C09149=1177.909,-61.811,-42.425,179.391,5.754,149.202
C09150=1177.904,-61.560,-42.436,179.394,5.755,149.202
C09151=1177.898,-61.311,-42.447,179.396,5.754,149.201
C09152=1177.894,-61.062,-42.458,179.398,5.755,149.201
C09153=1177.888,-60.811,-42.470,179.400,5.756,149.200
C09154=1177.883,-60.562,-42.481,179.403,5.756,149.199
C09155=1177.878,-60.313,-42.492,179.405,5.756,149.199
C09156=1177.872,-60.062,-42.503,179.407,5.756,149.198
C09157=1177.867,-59.813,-42.514,179.410,5.757,149.198
C09158=1177.862,-59.564,-42.525,179.412,5.757,149.197
C09159=1177.857,-59.314,-42.537,179.414,5.757,149.196
C09160=1177.851,-59.064,-42.547,179.417,5.758,149.196
C09161=1177.847,-58.815,-42.559,179.419,5.758,149.195
C09162=1177.841,-58.565,-42.570,179.421,5.758,149.194
C09163=1177.836,-58.314,-42.581,179.423,5.759,149.194
C09164=1177.831,-58.065,-42.592,179.426,5.759,149.193
C09165=1177.825,-57.815,-42.604,179.429,5.760,149.193
C09166=1177.821,-57.566,-42.615,179.430,5.760,149.192
C09167=1177.815,-57.316,-42.625,179.433,5.760,149.191
C09168=1177.810,-57.066,-42.637,179.436,5.761,149.191
C09169=1177.805,-56.817,-42.649,179.437,5.761,149.190
C09170=1177.800,-56.567,-42.660,179.440,5.761,149.189
C09171=1177.794,-56.318,-42.671,179.442,5.762,149.189
C09172=1177.789,-56.068,-42.682,179.445,5.762,149.188
C09173=1177.784,-55.818,-42.694,179.447,5.762,149.188
C09174=1177.779,-55.568,-42.705,179.449,5.763,149.187
C09175=1177.773,-55.319,-42.717,179.452,5.763,149.186
C09176=1177.768,-55.069,-42.728,179.454,5.763,149.186
C09177=1177.763,-54.819,-42.738,179.456,5.763,149.185
C09178=1177.758,-54.569,-42.750,179.459,5.764,149.185
C09179=1177.753,-54.320,-42.761,179.461,5.764,149.184
C09180=1177.747,-54.070,-42.773,179.464,5.765,149.183
C09181=1177.743,-53.821,-42.784,179.466,5.765,149.183
C09182=1177.737,-53.571,-42.796,179.468,5.765,149.182
C09183=1177.732,-53.322,-42.807,179.470,5.766,149.181
C09184=1177.726,-53.072,-42.819,179.473,5.766,149.181
C09185=1177.721,-52.821,-42.830,179.475,5.766,149.180
C09186=1177.717,-52.572,-42.841,179.477,5.767,149.180
C09187=1177.711,-52.322,-42.853,179.480,5.767,149.179
C09188=1177.706,-52.073,-42.864,179.482,5.767,149.178
C09189=1177.701,-51.823,-42.876,179.484,5.768,149.178
C09190=1177.696,-51.573,-42.887,179.487,5.768,149.177
C09191=1177.690,-51.324,-42.899,179.489,5.769,149.177
C09192=1177.686,-51.074,-42.910,179.492,5.769,149.176
C09193=1177.680,-50.825,-42.922,179.494,5.769,149.175
C09194=1177.674,-50.575,-42.934,179.496,5.770,149.175
C09195=1177.670,-50.325,-42.945,179.499,5.770,149.174
C09196=1177.664,-50.054,-42.957,179.501,5.771,149.173
C09197=1177.658,-49.784,-42.970,179.504,5.771,149.173
C09198=1177.652,-49.513,-42.982,179.506,5.771,149.172
C09199=1177.647,-49.244,-42.995,179.508,5.772,149.171
C09200=1177.642,-48.994,-43.006,179.511,5.772,149.171
C09201=1177.636,-48.744,-43.018,179.514,5.772,149.170
C09202=1177.631,-48.494,-43.030,179.516,5.773,149.169
C09203=1177.626,-48.245,-43.041,179.518,5.773,149.169
C09204=1177.621,-47.995,-43.053,179.521,5.773,149.168
C09205=1177.616,-47.746,-43.064,179.523,5.774,149.168
C09206=1177.610,-47.496,-43.076,179.525,5.774,149.167
C09207=1177.605,-47.246,-43.088,179.528,5.775,149.166
C09208=1177.600,-46.996,-43.099,179.530,5.775,149.166
C09209=1177.595,-46.746,-43.111,179.532,5.775,149.165
C09210=1177.590,-46.497,-43.122,179.535,5.776,149.164
C09211=1177.585,-46.247,-43.135,179.537,5.777,149.164
C09212=1177.579,-45.998,-43.146,179.539,5.776,149.163
C09213=1177.574,-45.749,-43.157,179.542,5.777,149.162
C09214=1177.569,-45.499,-43.169,179.544,5.777,149.162
C09215=1177.563,-45.249,-43.181,179.547,5.778,149.161
C09216=1177.559,-44.999,-43.192,179.549,5.778,149.161
C09217=1177.553,-44.749,-43.204,179.551,5.778,149.160
C09218=1177.548,-44.500,-43.216,179.554,5.779,149.159
C09219=1177.543,-44.250,-43.228,179.556,5.780,149.159
C09220=1177.538,-44.000,-43.240,179.559,5.780,149.158
C09221=1177.533,-43.751,-43.251,179.561,5.780,149.158
C09222=1177.527,-43.501,-43.263,179.563,5.780,149.157
C09223=1177.522,-43.251,-43.275,179.565,5.781,149.156
C09224=1177.516,-43.002,-43.287,179.568,5.781,149.156
C09225=1177.512,-42.753,-43.299,179.570,5.782,149.155
C09226=1177.506,-42.503,-43.311,179.572,5.782,149.154
C09227=1177.501,-42.253,-43.322,179.575,5.782,149.154
C09228=1177.496,-42.003,-43.334,179.577,5.783,149.153
C09229=1177.491,-41.753,-43.346,179.580,5.783,149.153
C09230=1177.486,-41.504,-43.358,179.583,5.784,149.152
C09231=1177.481,-41.254,-43.370,179.584,5.784,149.151
C09232=1177.476,-41.004,-43.381,179.587,5.784,149.151
C09233=1177.470,-40.754,-43.393,179.590,5.785,149.150
C09234=1177.465,-40.505,-43.406,179.592,5.786,149.150
C09235=1177.460,-40.255,-43.417,179.594,5.786,149.149
C09236=1177.455,-40.005,-43.429,179.596,5.786,149.148
C09237=1177.450,-39.755,-43.441,179.599,5.786,149.148
C09238=1177.444,-39.506,-43.454,179.601,5.787,149.147
C09239=1177.439,-39.257,-43.464,179.604,5.787,149.146
C09240=1177.434,-39.007,-43.476,179.606,5.788,149.146
C09241=1177.429,-38.758,-43.489,179.608,5.788,149.145
C09242=1177.423,-38.508,-43.501,179.611,5.788,149.144
C09243=1177.418,-38.258,-43.513,179.613,5.789,149.144
C09244=1177.413,-38.009,-43.525,179.616,5.789,149.143
C09245=1177.408,-37.759,-43.537,179.618,5.790,149.142
C09246=1177.402,-37.509,-43.549,179.620,5.790,149.142
C09247=1177.397,-37.260,-43.561,179.623,5.790,149.141
C09248=1177.392,-37.010,-43.573,179.625,5.791,149.141
C09249=1177.386,-36.760,-43.585,179.627,5.792,149.140
C09250=1177.382,-36.511,-43.597,179.630,5.792,149.139
C09251=1177.377,-36.261,-43.609,179.633,5.792,149.139
C09252=1177.372,-36.012,-43.621,179.634,5.792,149.138
C09253=1177.366,-35.762,-43.633,179.637,5.793,149.138
C09254=1177.361,-35.512,-43.645,179.640,5.793,149.137
C09255=1177.356,-35.263,-43.658,179.642,5.794,149.136
C09256=1177.351,-35.012,-43.669,179.645,5.795,149.136
C09257=1177.346,-34.763,-43.682,179.647,5.795,149.135
C09258=1177.341,-34.513,-43.694,179.649,5.795,149.135
C09259=1177.336,-34.264,-43.707,179.651,5.796,149.134
C09260=1177.330,-34.014,-43.718,179.654,5.796,149.133
C09261=1177.325,-33.764,-43.731,179.656,5.797,149.133
C09262=1177.320,-33.514,-43.743,179.659,5.797,149.132
C09263=1177.314,-33.265,-43.755,179.662,5.798,149.131
C09264=1177.309,-33.015,-43.767,179.663,5.798,149.131
C09265=1177.305,-32.766,-43.779,179.666,5.798,149.130
C09266=1177.299,-32.516,-43.791,179.669,5.799,149.129
C09267=1177.294,-32.266,-43.803,179.671,5.799,149.129
C09268=1177.289,-32.017,-43.816,179.673,5.800,149.128
C09269=1177.284,-31.768,-43.828,179.676,5.800,149.128
C09270=1177.278,-31.518,-43.840,179.678,5.800,149.127
C09271=1177.273,-31.268,-43.853,179.680,5.801,149.126
C09272=1177.268,-31.018,-43.865,179.683,5.801,149.126
C09273=1177.263,-30.769,-43.878,179.685,5.802,149.125
C09274=1177.258,-30.519,-43.890,179.688,5.802,149.125
C09275=1177.253,-30.269,-43.902,179.690,5.803,149.124
C09276=1177.247,-30.019,-43.914,179.693,5.804,149.123
C09277=1177.242,-29.770,-43.927,179.695,5.803,149.123
C09278=1177.237,-29.521,-43.939,179.697,5.804,149.122
C09279=1177.232,-29.271,-43.951,179.700,5.805,149.121
C09280=1177.226,-29.021,-43.964,179.702,5.805,149.121
C09281=1177.222,-28.771,-43.977,179.705,5.805,149.120
C09282=1177.217,-28.521,-43.989,179.707,5.806,149.120
C09283=1177.211,-28.272,-44.001,179.710,5.807,149.119
C09284=1177.206,-28.022,-44.013,179.712,5.806,149.118
C09285=1177.201,-27.773,-44.026,179.714,5.807,149.118
C09286=1177.196,-27.524,-44.038,179.717,5.808,149.117
C09287=1177.190,-27.274,-44.050,179.719,5.808,149.116
C09288=1177.186,-27.024,-44.063,179.721,5.809,149.116
C09289=1177.181,-26.774,-44.076,179.724,5.809,149.115
C09290=1177.175,-26.524,-44.088,179.727,5.810,149.114
C09291=1177.170,-26.275,-44.100,179.728,5.810,149.114
C09292=1177.165,-26.026,-44.113,179.731,5.810,149.113
C09293=1177.160,-25.776,-44.125,179.734,5.811,149.113
C09294=1177.155,-25.526,-44.138,179.736,5.812,149.112
C09295=1177.150,-25.276,-44.150,179.739,5.812,149.111
C09296=1177.145,-25.027,-44.163,179.741,5.812,149.111
C09297=1177.140,-24.778,-44.175,179.743,5.813,149.110
C09298=1177.133,-24.528,-44.188,179.746,5.814,149.110
C09299=1177.129,-24.278,-44.201,179.748,5.813,149.109
C09300=1177.123,-24.009,-44.214,179.751,5.814,149.108
C09301=1177.118,-23.739,-44.228,179.753,5.815,149.108
C09302=1177.112,-23.469,-44.241,179.756,5.816,149.107
C09303=1177.107,-23.199,-44.255,179.759,5.816,149.106
C09304=1177.102,-22.950,-44.267,179.761,5.816,149.106
C09305=1177.097,-22.700,-44.280,179.764,5.816,149.105
C09306=1177.091,-22.450,-44.293,179.766,5.817,149.104
C09307=1177.086,-22.200,-44.305,179.768,5.818,149.104
C09308=1177.081,-21.951,-44.318,179.771,5.818,149.103
C09309=1177.076,-21.702,-44.331,179.773,5.819,149.103
C09310=1177.071,-21.452,-44.344,179.776,5.819,149.102
C09311=1177.066,-21.202,-44.356,179.779,5.820,149.101
C09312=1177.060,-20.953,-44.369,179.781,5.821,149.101
C09313=1177.055,-20.703,-44.381,179.783,5.820,149.100
C09314=1177.050,-20.453,-44.394,179.785,5.821,149.099
C09315=1177.045,-20.203,-44.407,179.788,5.822,149.099
C09316=1177.040,-19.954,-44.419,179.790,5.822,149.098
C09317=1177.034,-19.704,-44.433,179.793,5.822,149.098
C09318=1177.029,-19.454,-44.446,179.795,5.823,149.097
C09319=1177.024,-19.205,-44.458,179.798,5.824,149.096
C09320=1177.019,-18.956,-44.471,179.800,5.824,149.096
C09321=1177.014,-18.706,-44.483,179.803,5.825,149.095
C09322=1177.009,-18.456,-44.497,179.805,5.825,149.094
C09323=1177.004,-18.207,-44.510,179.807,5.825,149.094
C09324=1176.999,-17.957,-44.522,179.810,5.826,149.093
C09325=1176.994,-17.707,-44.535,179.812,5.826,149.093
C09326=1176.988,-17.458,-44.548,179.815,5.827,149.092
C09327=1176.983,-17.208,-44.560,179.817,5.828,149.091
C09328=1176.978,-16.958,-44.573,179.820,5.828,149.091
C09329=1176.973,-16.709,-44.586,179.822,5.829,149.090
C09330=1176.967,-16.459,-44.599,179.825,5.829,149.090
C09331=1176.962,-16.210,-44.612,179.827,5.830,149.089
C09332=1176.958,-15.960,-44.625,179.830,5.830,149.088
C09333=1176.952,-15.711,-44.638,179.832,5.831,149.088
C09334=1176.947,-15.461,-44.651,179.835,5.832,149.087
C09335=1176.942,-15.211,-44.664,179.837,5.831,149.086
C09336=1176.937,-14.962,-44.677,179.839,5.832,149.086
C09337=1176.931,-14.712,-44.690,179.842,5.833,149.085
C09338=1176.927,-14.462,-44.703,179.844,5.833,149.085
C09339=1176.922,-14.213,-44.715,179.846,5.834,149.084
C09340=1176.916,-13.963,-44.729,179.849,5.834,149.083
C09341=1176.911,-13.713,-44.742,179.852,5.835,149.083
C09342=1176.906,-13.464,-44.754,179.854,5.836,149.082
C09343=1176.900,-13.214,-44.767,179.857,5.836,149.082
C09344=1176.896,-12.964,-44.780,179.859,5.836,149.081
C09345=1176.890,-12.715,-44.794,179.861,5.837,149.080
C09346=1176.886,-12.465,-44.807,179.864,5.838,149.080
C09347=1176.881,-12.216,-44.820,179.867,5.838,149.079
C09348=1176.875,-11.966,-44.833,179.869,5.839,149.079
C09349=1176.870,-11.716,-44.846,179.872,5.840,149.078
C09350=1176.865,-11.467,-44.859,179.874,5.840,149.077
C09351=1176.860,-11.217,-44.873,179.876,5.840,149.077
C09352=1176.855,-10.968,-44.885,179.878,5.840,149.076
C09353=1176.849,-10.718,-44.899,179.881,5.841,149.075
C09354=1176.845,-10.468,-44.912,179.883,5.842,149.075
C09355=1176.840,-10.219,-44.924,179.886,5.842,149.074
C09356=1176.835,-9.969,-44.938,179.889,5.843,149.073
C09357=1176.829,-9.720,-44.951,179.891,5.843,149.073
C09358=1176.824,-9.470,-44.964,179.893,5.844,149.072
C09359=1176.819,-9.220,-44.977,179.896,5.844,149.072
C09360=1176.814,-8.971,-44.991,179.898,5.845,149.071
C09361=1176.809,-8.721,-45.004,179.901,5.846,149.070
C09362=1176.804,-8.472,-45.017,179.904,5.846,149.070
C09363=1176.799,-8.222,-45.030,179.906,5.847,149.069
C09364=1176.794,-7.973,-45.044,179.908,5.847,149.069
C09365=1176.788,-7.723,-45.057,179.911,5.848,149.068
C09366=1176.783,-7.473,-45.070,179.913,5.849,149.067
C09367=1176.778,-7.224,-45.084,179.916,5.849,149.067
C09368=1176.773,-6.974,-45.097,179.919,5.850,149.066
C09369=1176.767,-6.725,-45.110,179.921,5.851,149.066
C09370=1176.763,-6.475,-45.124,179.923,5.851,149.065
C09371=1176.757,-6.226,-45.137,179.926,5.851,149.064
C09372=1176.753,-5.976,-45.150,179.929,5.852,149.063
C09373=1176.747,-5.727,-45.164,179.931,5.853,149.063
C09374=1176.743,-5.477,-45.177,179.934,5.853,149.062
C09375=1176.737,-5.227,-45.190,179.936,5.854,149.062
C09376=1176.733,-4.978,-45.203,179.938,5.854,149.061
C09377=1176.727,-4.728,-45.217,179.940,5.854,149.060
C09378=1176.722,-4.478,-45.230,179.943,5.855,149.060
C09379=1176.717,-4.229,-45.244,179.945,5.855,149.059
C09380=1176.712,-3.979,-45.257,179.948,5.856,149.059
C09381=1176.707,-3.730,-45.270,179.951,5.856,149.058
C09382=1176.701,-3.480,-45.284,179.953,5.857,149.057
C09383=1176.697,-3.231,-45.297,179.955,5.858,149.057
C09384=1176.691,-2.981,-45.311,179.958,5.858,149.056
C09385=1176.686,-2.731,-45.323,179.960,5.859,149.056
C09386=1176.681,-2.482,-45.338,179.963,5.859,149.055
C09387=1176.675,-2.232,-45.351,179.965,5.860,149.055
C09388=1176.671,-1.982,-45.365,179.968,5.861,149.054
C09389=1176.665,-1.733,-45.378,179.970,5.861,149.053
C09390=1176.660,-1.483,-45.392,179.972,5.862,149.053
C09391=1176.655,-1.234,-45.405,179.975,5.863,149.052
C09392=1176.650,-0.984,-45.419,179.978,5.863,149.051
C09393=1176.645,-0.735,-45.432,179.980,5.864,149.051
C09394=1176.640,-0.485,-45.446,179.983,5.864,149.050
C09395=1176.635,-0.235,-45.459,179.985,5.865,149.049
C09396=1176.630,0.014,-45.473,179.987,5.866,149.049
C09397=1176.625,0.264,-45.487,179.990,5.866,149.048
C09398=1176.619,0.513,-45.500,179.993,5.867,149.048
C09399=1176.615,0.763,-45.514,179.995,5.867,149.047
C09400=1176.609,1.012,-45.527,179.998,5.868,149.046
C09401=1176.604,1.262,-45.541,-180.000,5.868,149.046
C09402=1176.600,1.512,-45.554,-179.998,5.869,149.045
C09403=1176.594,1.761,-45.568,-179.995,5.870,149.045
C09404=1176.589,2.030,-45.583,-179.992,5.871,149.044
C09405=1176.583,2.300,-45.598,-179.989,5.871,149.043
C09406=1176.577,2.569,-45.613,-179.986,5.872,149.043
C09407=1176.572,2.838,-45.628,-179.984,5.872,149.042
C09408=1176.567,3.088,-45.641,-179.982,5.873,149.041
C09409=1176.562,3.337,-45.655,-179.979,5.874,149.041
C09410=1176.557,3.587,-45.669,-179.976,5.874,149.040
C09411=1176.552,3.837,-45.683,-179.974,5.875,149.040
C09412=1176.547,4.086,-45.696,-179.971,5.875,149.039
C09413=1176.542,4.335,-45.710,-179.969,5.876,149.038
C09414=1176.537,4.586,-45.724,-179.967,5.877,149.038
C09415=1176.531,4.835,-45.738,-179.964,5.877,149.037
C09416=1176.527,5.084,-45.751,-179.961,5.878,149.036
C09417=1176.521,5.333,-45.765,-179.959,5.878,149.036
C09418=1176.516,5.584,-45.779,-179.956,5.879,149.035
C09419=1176.511,5.833,-45.793,-179.954,5.879,149.035
C09420=1176.506,6.082,-45.806,-179.952,5.880,149.034
C09421=1176.501,6.332,-45.821,-179.949,5.881,149.033
C09422=1176.496,6.582,-45.834,-179.947,5.882,149.033
C09423=1176.490,6.831,-45.848,-179.944,5.883,149.032
C09424=1176.485,7.081,-45.862,-179.941,5.883,149.032
C09425=1176.481,7.330,-45.877,-179.939,5.884,149.031
C09426=1176.475,7.580,-45.889,-179.936,5.885,149.030
C09427=1176.470,7.829,-45.904,-179.933,5.885,149.030
C09428=1176.465,8.079,-45.918,-179.931,5.886,149.029
C09429=1176.461,8.329,-45.932,-179.929,5.886,149.029
C09430=1176.455,8.578,-45.946,-179.926,5.887,149.028
C09431=1176.450,8.828,-45.960,-179.924,5.888,149.027
C09432=1176.446,9.078,-45.973,-179.921,5.888,149.027
C09433=1176.440,9.327,-45.987,-179.919,5.889,149.026
C09434=1176.435,9.576,-46.001,-179.916,5.890,149.026
C09435=1176.430,9.826,-46.016,-179.914,5.890,149.025
C09436=1176.425,10.076,-46.030,-179.911,5.890,149.024
C09437=1176.420,10.325,-46.044,-179.909,5.891,149.024
C09438=1176.415,10.574,-46.058,-179.906,5.892,149.023
C09439=1176.410,10.824,-46.072,-179.904,5.892,149.022
C09440=1176.404,11.073,-46.086,-179.901,5.893,149.022
C09441=1176.399,11.324,-46.100,-179.899,5.894,149.021
C09442=1176.395,11.573,-46.114,-179.896,5.895,149.021
C09443=1176.390,11.823,-46.128,-179.893,5.896,149.020
C09444=1176.384,12.072,-46.142,-179.891,5.896,149.019
C09445=1176.379,12.321,-46.156,-179.889,5.897,149.019
C09446=1176.374,12.571,-46.170,-179.886,5.897,149.018
C09447=1176.369,12.821,-46.185,-179.883,5.898,149.018
C09448=1176.364,13.070,-46.199,-179.881,5.899,149.017
C09449=1176.359,13.320,-46.213,-179.878,5.899,149.016
C09450=1176.354,13.569,-46.227,-179.876,5.900,149.016
C09451=1176.349,13.819,-46.241,-179.874,5.901,149.015
C09452=1176.344,14.069,-46.256,-179.871,5.901,149.015
C09453=1176.338,14.318,-46.270,-179.868,5.902,149.014
C09454=1176.333,14.567,-46.284,-179.866,5.902,149.014
C09455=1176.328,14.817,-46.298,-179.863,5.904,149.013
C09456=1176.323,15.067,-46.312,-179.860,5.904,149.012
C09457=1176.318,15.316,-46.327,-179.858,5.905,149.012
C09458=1176.313,15.565,-46.341,-179.855,5.906,149.011
C09459=1176.308,15.815,-46.355,-179.853,5.906,149.010
C09460=1176.303,16.064,-46.370,-179.851,5.907,149.010
C09461=1176.298,16.314,-46.384,-179.848,5.907,149.009
C09462=1176.293,16.564,-46.398,-179.846,5.908,149.009
C09463=1176.288,16.813,-46.412,-179.843,5.909,149.008
C09464=1176.283,17.062,-46.427,-179.841,5.909,149.007
C09465=1176.278,17.312,-46.441,-179.838,5.910,149.007
C09466=1176.272,17.562,-46.456,-179.835,5.911,149.006
C09467=1176.267,17.812,-46.470,-179.832,5.912,149.006
C09468=1176.263,18.061,-46.485,-179.830,5.913,149.005
C09469=1176.258,18.311,-46.499,-179.828,5.913,149.004
C09470=1176.252,18.560,-46.513,-179.825,5.914,149.004
C09471=1176.247,18.809,-46.527,-179.823,5.914,149.003
C09472=1176.242,19.059,-46.542,-179.820,5.915,149.003
C09473=1176.237,19.309,-46.556,-179.818,5.916,149.002
C09474=1176.233,19.558,-46.571,-179.815,5.916,149.001
C09475=1176.228,19.808,-46.585,-179.813,5.917,149.001
C09476=1176.222,20.058,-46.600,-179.810,5.918,149.000
C09477=1176.216,20.307,-46.614,-179.807,5.919,149.000
C09478=1176.212,20.556,-46.629,-179.805,5.919,148.999
C09479=1176.207,20.805,-46.643,-179.803,5.920,148.998
C09480=1176.202,21.055,-46.658,-179.800,5.921,148.998
C09481=1176.197,21.305,-46.672,-179.797,5.921,148.997
C09482=1176.192,21.554,-46.687,-179.795,5.922,148.997
C09483=1176.187,21.804,-46.702,-179.792,5.922,148.996
C09484=1176.182,22.054,-46.716,-179.790,5.924,148.996
C09485=1176.177,22.303,-46.730,-179.787,5.925,148.995
C09486=1176.172,22.553,-46.745,-179.784,5.925,148.994
C09487=1176.167,22.802,-46.760,-179.782,5.926,148.994
C09488=1176.161,23.052,-46.774,-179.780,5.926,148.993
C09489=1176.156,23.301,-46.789,-179.777,5.927,148.992
C09490=1176.151,23.550,-46.803,-179.775,5.928,148.992
C09491=1176.146,23.800,-46.818,-179.772,5.928,148.991
C09492=1176.142,24.049,-46.833,-179.769,5.930,148.991
C09493=1176.136,24.299,-46.847,-179.767,5.930,148.990
C09494=1176.131,24.548,-46.862,-179.764,5.931,148.989
C09495=1176.126,24.798,-46.877,-179.762,5.932,148.989
C09496=1176.121,25.048,-46.891,-179.759,5.932,148.988
C09497=1176.116,25.297,-46.907,-179.757,5.933,148.988
C09498=1176.111,25.547,-46.921,-179.754,5.934,148.987
C09499=1176.106,25.796,-46.936,-179.751,5.935,148.986
C09500=1176.101,26.046,-46.950,-179.749,5.935,148.986
C09501=1176.096,26.296,-46.965,-179.746,5.936,148.985
C09502=1176.091,26.545,-46.980,-179.744,5.937,148.985
C09503=1176.086,26.794,-46.994,-179.742,5.938,148.984
C09504=1176.081,27.044,-47.010,-179.739,5.938,148.984
C09505=1176.076,27.294,-47.024,-179.736,5.939,148.983
C09506=1176.071,27.543,-47.039,-179.734,5.940,148.982
C09507=1176.065,27.793,-47.054,-179.731,5.941,148.982
C09508=1176.060,28.061,-47.070,-179.728,5.941,148.981
C09509=1176.055,28.330,-47.085,-179.726,5.942,148.980
C09510=1176.049,28.599,-47.102,-179.723,5.943,148.980
C09511=1176.044,28.867,-47.118,-179.720,5.944,148.979
C09512=1176.039,29.118,-47.133,-179.718,5.944,148.979
C09513=1176.034,29.367,-47.148,-179.715,5.945,148.978
C09514=1176.029,29.616,-47.162,-179.712,5.946,148.977
C09515=1176.024,29.866,-47.178,-179.710,5.947,148.977
C09516=1176.019,30.115,-47.192,-179.707,5.948,148.976
C09517=1176.014,30.365,-47.207,-179.705,5.948,148.976
C09518=1176.009,30.614,-47.223,-179.702,5.949,148.975
C09519=1176.004,30.864,-47.237,-179.700,5.950,148.975
C09520=1175.998,31.113,-47.253,-179.697,5.951,148.974
C09521=1175.993,31.363,-47.267,-179.695,5.952,148.973
C09522=1175.989,31.612,-47.282,-179.692,5.952,148.973
C09523=1175.983,31.861,-47.298,-179.689,5.953,148.972
C09524=1175.978,32.111,-47.312,-179.687,5.954,148.972
C09525=1175.973,32.360,-47.327,-179.684,5.955,148.971
C09526=1175.969,32.610,-47.343,-179.682,5.956,148.970
C09527=1175.963,32.860,-47.358,-179.679,5.956,148.970
C09528=1175.959,33.109,-47.373,-179.676,5.957,148.969
C09529=1175.953,33.359,-47.388,-179.674,5.958,148.969
C09530=1175.948,33.608,-47.402,-179.672,5.958,148.968
C09531=1175.944,33.857,-47.417,-179.669,5.960,148.968
C09532=1175.938,34.107,-47.433,-179.666,5.960,148.967
C09533=1175.933,34.357,-47.447,-179.664,5.961,148.966
C09534=1175.928,34.606,-47.463,-179.661,5.962,148.966
C09535=1175.923,34.855,-47.478,-179.659,5.962,148.965
C09536=1175.919,35.105,-47.494,-179.656,5.964,148.965
C09537=1175.914,35.355,-47.508,-179.653,5.964,148.964
C09538=1175.908,35.604,-47.524,-179.651,5.965,148.963
C09539=1175.904,35.853,-47.539,-179.649,5.966,148.963
C09540=1175.898,36.103,-47.554,-179.646,5.966,148.962
C09541=1175.894,36.352,-47.569,-179.643,5.968,148.962
C09542=1175.888,36.602,-47.584,-179.641,5.968,148.961
C09543=1175.883,36.852,-47.600,-179.638,5.969,148.960
C09544=1175.878,37.101,-47.615,-179.636,5.970,148.960
C09545=1175.873,37.350,-47.631,-179.632,5.971,148.959
C09546=1175.868,37.600,-47.646,-179.630,5.972,148.959
C09547=1175.863,37.850,-47.661,-179.628,5.972,148.958
C09548=1175.858,38.099,-47.676,-179.625,5.973,148.957
C09549=1175.853,38.349,-47.692,-179.623,5.974,148.957
C09550=1175.848,38.598,-47.707,-179.620,5.975,148.956
C09551=1175.843,38.847,-47.722,-179.618,5.976,148.956
C09552=1175.838,39.097,-47.738,-179.615,5.976,148.955
C09553=1175.833,39.346,-47.753,-179.612,5.977,148.955
C09554=1175.828,39.595,-47.768,-179.610,5.978,148.954
C09555=1175.823,39.845,-47.784,-179.607,5.979,148.953
C09556=1175.818,40.095,-47.798,-179.605,5.980,148.953
C09557=1175.813,40.344,-47.814,-179.602,5.980,148.952
C09558=1175.807,40.594,-47.830,-179.599,5.981,148.952
C09559=1175.803,40.843,-47.845,-179.597,5.983,148.951
C09560=1175.798,41.093,-47.861,-179.594,5.983,148.950
C09561=1175.792,41.342,-47.876,-179.592,5.984,148.950
C09562=1175.788,41.591,-47.891,-179.589,5.984,148.949
C09563=1175.782,41.841,-47.907,-179.586,5.986,148.949
C09564=1175.778,42.091,-47.923,-179.584,5.987,148.948
C09565=1175.773,42.340,-47.938,-179.581,5.987,148.948
C09566=1175.768,42.589,-47.953,-179.579,5.988,148.947
C09567=1175.762,42.839,-47.969,-179.576,5.989,148.946
C09568=1175.758,43.089,-47.984,-179.574,5.990,148.946
C09569=1175.753,43.338,-48.000,-179.571,5.991,148.945
C09570=1175.747,43.587,-48.015,-179.568,5.991,148.945
C09571=1175.743,43.837,-48.030,-179.566,5.993,148.944
C09572=1175.738,44.087,-48.046,-179.563,5.993,148.944
C09573=1175.733,44.335,-48.063,-179.561,5.994,148.943
C09574=1175.727,44.585,-48.078,-179.558,5.995,148.942
C09575=1175.723,44.834,-48.093,-179.555,5.996,148.942
C09576=1175.718,45.084,-48.109,-179.553,5.997,148.941
C09577=1175.713,45.333,-48.125,-179.550,5.997,148.941
C09578=1175.707,45.583,-48.140,-179.548,5.998,148.940
C09579=1175.703,45.833,-48.156,-179.545,6.000,148.940
C09580=1175.698,46.082,-48.171,-179.543,6.000,148.939
C09581=1175.692,46.331,-48.187,-179.540,6.001,148.938
C09582=1175.688,46.581,-48.204,-179.537,6.001,148.938
C09583=1175.683,46.830,-48.219,-179.535,6.003,148.937
C09584=1175.678,47.079,-48.234,-179.532,6.004,148.937
C09585=1175.673,47.330,-48.250,-179.530,6.005,148.936
C09586=1175.668,47.579,-48.266,-179.527,6.005,148.936
C09587=1175.663,47.828,-48.282,-179.524,6.007,148.935
C09588=1175.658,48.078,-48.298,-179.522,6.007,148.934
C09589=1175.653,48.327,-48.313,-179.519,6.008,148.934
C09590=1175.648,48.576,-48.329,-179.516,6.009,148.933
C09591=1175.643,48.826,-48.345,-179.514,6.010,148.933
C09592=1175.638,49.075,-48.361,-179.512,6.011,148.932
C09593=1175.633,49.325,-48.376,-179.509,6.011,148.932
C09594=1175.628,49.575,-48.392,-179.506,6.013,148.931
C09595=1175.623,49.824,-48.409,-179.504,6.013,148.930
C09596=1175.618,50.073,-48.424,-179.501,6.014,148.930
C09597=1175.613,50.323,-48.440,-179.498,6.016,148.929
C09598=1175.608,50.572,-48.455,-179.496,6.016,148.929
C09599=1175.603,50.822,-48.472,-179.493,6.017,148.928
C09600=1175.598,51.071,-48.487,-179.491,6.018,148.928
C09601=1175.593,51.320,-48.503,-179.488,6.019,148.927
C09602=1175.588,51.570,-48.520,-179.485,6.020,148.926
C09603=1175.583,51.819,-48.535,-179.483,6.021,148.926
C09604=1175.578,52.069,-48.551,-179.480,6.022,148.925
C09605=1175.573,52.318,-48.568,-179.477,6.022,148.925
C09606=1175.568,52.567,-48.583,-179.475,6.023,148.924
C09607=1175.564,52.817,-48.599,-179.472,6.025,148.924
C09608=1175.558,53.066,-48.615,-179.470,6.026,148.923
C09609=1175.554,53.316,-48.631,-179.467,6.026,148.922
C09610=1175.549,53.565,-48.647,-179.465,6.028,148.922
C09611=1175.544,53.815,-48.663,-179.462,6.028,148.921
C09612=1175.538,54.084,-48.680,-179.459,6.029,148.921
C09613=1175.533,54.351,-48.698,-179.457,6.030,148.920
C09614=1175.527,54.620,-48.715,-179.454,6.031,148.920
C09615=1175.522,54.889,-48.732,-179.451,6.032,148.919
C09616=1175.517,55.138,-48.748,-179.449,6.033,148.918
C09617=1175.513,55.388,-48.764,-179.446,6.034,148.918
C09618=1175.507,55.637,-48.781,-179.443,6.035,148.917
C09619=1175.501,55.887,-48.797,-179.440,6.036,148.917
C09620=1175.497,56.136,-48.814,-179.438,6.036,148.916
C09621=1175.491,56.385,-48.829,-179.435,6.038,148.916
C09622=1175.487,56.635,-48.846,-179.432,6.039,148.915
C09623=1175.482,56.884,-48.861,-179.430,6.039,148.914
C09624=1175.477,57.134,-48.878,-179.427,6.041,148.914
C09625=1175.472,57.383,-48.894,-179.425,6.042,148.913
C09626=1175.467,57.633,-48.910,-179.422,6.042,148.913
C09627=1175.462,57.882,-48.926,-179.420,6.044,148.912
C09628=1175.457,58.132,-48.943,-179.417,6.044,148.912
C09629=1175.452,58.380,-48.959,-179.415,6.045,148.911
C09630=1175.448,58.630,-48.975,-179.412,6.047,148.911
C09631=1175.442,58.879,-48.991,-179.409,6.047,148.910
C09632=1175.437,59.130,-49.008,-179.407,6.048,148.909
C09633=1175.432,59.378,-49.024,-179.404,6.049,148.909
C09634=1175.427,59.628,-49.041,-179.401,6.050,148.908
C09635=1175.423,59.878,-49.057,-179.399,6.051,148.908
C09636=1175.417,60.127,-49.073,-179.396,6.052,148.907
C09637=1175.413,60.376,-49.090,-179.393,6.053,148.907
C09638=1175.408,60.626,-49.105,-179.391,6.055,148.906
C09639=1175.403,60.875,-49.122,-179.388,6.055,148.905
C09640=1175.397,61.124,-49.139,-179.386,6.056,148.905
C09641=1175.393,61.374,-49.155,-179.383,6.057,148.904
C09642=1175.387,61.623,-49.171,-179.381,6.058,148.904
C09643=1175.383,61.873,-49.188,-179.378,6.059,148.903
C09644=1175.378,62.122,-49.204,-179.375,6.060,148.903
C09645=1175.372,62.372,-49.221,-179.373,6.061,148.902
C09646=1175.368,62.621,-49.237,-179.370,6.062,148.902
C09647=1175.363,62.870,-49.254,-179.367,6.063,148.901
C09648=1175.358,63.120,-49.270,-179.365,6.064,148.901
C09649=1175.354,63.370,-49.286,-179.362,6.065,148.900
C09650=1175.348,63.619,-49.303,-179.360,6.066,148.900
C09651=1175.343,63.868,-49.320,-179.357,6.067,148.899
C09652=1175.338,64.117,-49.336,-179.354,6.068,148.898
C09653=1175.334,64.367,-49.353,-179.352,6.069,148.898
C09654=1175.328,64.617,-49.369,-179.349,6.069,148.897
C09655=1175.323,64.866,-49.386,-179.346,6.071,148.897
C09656=1175.319,65.115,-49.402,-179.344,6.072,148.896
C09657=1175.314,65.364,-49.419,-179.341,6.073,148.896
C09658=1175.308,65.614,-49.436,-179.338,6.074,148.895
C09659=1175.304,65.863,-49.452,-179.336,6.075,148.894
C09660=1175.299,66.112,-49.469,-179.333,6.076,148.894
C09661=1175.294,66.362,-49.485,-179.331,6.077,148.893
C09662=1175.289,66.612,-49.502,-179.328,6.077,148.893
C09663=1175.284,66.861,-49.518,-179.325,6.079,148.892
C09664=1175.279,67.110,-49.535,-179.323,6.080,148.892
C09665=1175.274,67.360,-49.552,-179.320,6.081,148.891
C09666=1175.269,67.609,-49.568,-179.317,6.082,148.891
C09667=1175.264,67.858,-49.585,-179.315,6.083,148.890
C09668=1175.259,68.108,-49.602,-179.312,6.084,148.889
C09669=1175.254,68.357,-49.619,-179.310,6.085,148.889
C09670=1175.250,68.606,-49.635,-179.307,6.086,148.888
C09671=1175.244,68.856,-49.653,-179.305,6.087,148.888
C09672=1175.240,69.106,-49.669,-179.302,6.088,148.887
C09673=1175.235,69.354,-49.686,-179.299,6.089,148.887
C09674=1175.230,69.604,-49.703,-179.297,6.090,148.886
C09675=1175.225,69.854,-49.720,-179.294,6.092,148.886
C09676=1175.219,70.103,-49.736,-179.291,6.092,148.885
C09677=1175.215,70.352,-49.753,-179.288,6.094,148.885
C09678=1175.210,70.602,-49.770,-179.286,6.094,148.884
C09679=1175.205,70.851,-49.787,-179.284,6.095,148.884
C09680=1175.200,71.100,-49.803,-179.280,6.097,148.883
C09681=1175.195,71.350,-49.821,-179.278,6.097,148.882
C09682=1175.190,71.600,-49.837,-179.276,6.099,148.882
C09683=1175.185,71.848,-49.855,-179.273,6.100,148.881
C09684=1175.180,72.098,-49.872,-179.270,6.101,148.881
C09685=1175.175,72.347,-49.889,-179.268,6.102,148.880
C09686=1175.171,72.597,-49.906,-179.265,6.103,148.880
C09687=1175.166,72.846,-49.922,-179.262,6.104,148.879
C09688=1175.160,73.095,-49.939,-179.260,6.105,148.879
C09689=1175.156,73.345,-49.956,-179.257,6.106,148.878
C09690=1175.151,73.595,-49.973,-179.255,6.107,148.878
C09691=1175.146,73.844,-49.990,-179.252,6.109,148.877
C09692=1175.141,74.093,-50.007,-179.249,6.109,148.877
C09693=1175.136,74.342,-50.024,-179.247,6.110,148.876
C09694=1175.131,74.592,-50.041,-179.244,6.112,148.876
C09695=1175.126,74.841,-50.058,-179.241,6.112,148.875
C09696=1175.121,75.090,-50.076,-179.239,6.114,148.874
C09697=1175.117,75.339,-50.092,-179.236,6.114,148.874
C09698=1175.111,75.589,-50.109,-179.233,6.116,148.873
C09699=1175.106,75.839,-50.127,-179.231,6.117,148.873
C09700=1175.102,76.088,-50.144,-179.228,6.118,148.872
C09701=1175.097,76.338,-50.161,-179.225,6.119,148.872
C09702=1175.092,76.586,-50.178,-179.223,6.120,148.871
C09703=1175.087,76.836,-50.196,-179.220,6.121,148.871
C09704=1175.082,77.085,-50.212,-179.218,6.122,148.870
C09705=1175.077,77.335,-50.230,-179.215,6.124,148.870
C09706=1175.072,77.585,-50.247,-179.212,6.124,148.869
C09707=1175.068,77.834,-50.264,-179.210,6.126,148.869
C09708=1175.062,78.083,-50.281,-179.207,6.126,148.868
C09709=1175.057,78.332,-50.298,-179.204,6.128,148.868
C09710=1175.052,78.581,-50.316,-179.202,6.129,148.867
C09711=1175.047,78.831,-50.333,-179.199,6.130,148.866
C09712=1175.043,79.080,-50.350,-179.196,6.131,148.866
C09713=1175.038,79.330,-50.368,-179.194,6.133,148.865
C09714=1175.033,79.580,-50.385,-179.191,6.133,148.865
C09715=1175.028,79.828,-50.402,-179.189,6.134,148.864
C09716=1175.022,80.097,-50.421,-179.186,6.135,148.864
C09717=1175.017,80.365,-50.439,-179.183,6.137,148.863
C09718=1175.012,80.634,-50.459,-179.180,6.138,148.863
C09719=1175.007,80.902,-50.477,-179.178,6.139,148.862
C09720=1175.002,81.151,-50.494,-179.174,6.141,148.862
C09721=1174.997,81.401,-50.512,-179.172,6.142,148.861
C09722=1174.992,81.650,-50.528,-179.169,6.143,148.860
C09723=1174.987,81.899,-50.546,-179.167,6.144,148.860
C09724=1174.982,82.149,-50.564,-179.164,6.145,148.859
C09725=1174.977,82.398,-50.582,-179.162,6.146,148.859
C09726=1174.973,82.648,-50.598,-179.158,6.147,148.858
C09727=1174.968,82.897,-50.616,-179.156,6.148,148.858
C09728=1174.963,83.146,-50.634,-179.154,6.150,148.857
C09729=1174.958,83.395,-50.651,-179.151,6.150,148.857
C09730=1174.953,83.644,-50.669,-179.148,6.152,148.856
C09731=1174.948,83.894,-50.686,-179.146,6.153,148.856
C09732=1174.943,84.143,-50.704,-179.143,6.154,148.855
C09733=1174.937,84.393,-50.721,-179.140,6.155,148.855
C09734=1174.933,84.642,-50.738,-179.137,6.157,148.854
C09735=1174.928,84.891,-50.756,-179.135,6.157,148.854
C09736=1174.923,85.141,-50.774,-179.132,6.159,148.853
C09737=1174.918,85.390,-50.792,-179.130,6.160,148.853
C09738=1174.913,85.640,-50.809,-179.127,6.161,148.852
C09739=1174.909,85.888,-50.826,-179.125,6.162,148.852
C09740=1174.904,86.138,-50.844,-179.121,6.163,148.851
C09741=1174.899,86.387,-50.862,-179.119,6.164,148.851
C09742=1174.894,86.637,-50.880,-179.117,6.166,148.850
C09743=1174.889,86.886,-50.898,-179.114,6.167,148.849
C09744=1174.884,87.135,-50.915,-179.111,6.168,148.849
C09745=1174.879,87.384,-50.932,-179.109,6.169,148.848
C09746=1174.875,87.634,-50.950,-179.106,6.170,148.848
C09747=1174.870,87.883,-50.968,-179.103,6.171,148.847
C09748=1174.864,88.133,-50.985,-179.101,6.173,148.847
C09749=1174.859,88.382,-51.003,-179.098,6.174,148.847
C09750=1174.855,88.631,-51.021,-179.095,6.175,148.846
C09751=1174.850,88.880,-51.039,-179.093,6.176,148.845
C09752=1174.844,89.130,-51.057,-179.090,6.177,148.845
C09753=1174.840,89.379,-51.075,-179.087,6.179,148.844
C09754=1174.836,89.629,-51.092,-179.085,6.180,148.844
C09755=1174.831,89.878,-51.110,-179.082,6.181,148.843
C09756=1174.826,90.128,-51.128,-179.080,6.182,148.843
C09757=1174.821,90.377,-51.146,-179.076,6.183,148.842
C09758=1174.816,90.626,-51.164,-179.074,6.184,148.842
C09759=1174.811,90.875,-51.182,-179.072,6.186,148.841
C09760=1174.806,91.124,-51.200,-179.069,6.187,148.841
C09761=1174.801,91.373,-51.217,-179.066,6.188,148.840
C09762=1174.796,91.623,-51.235,-179.064,6.189,148.840
C09763=1174.791,91.872,-51.253,-179.061,6.191,148.839
C09764=1174.786,92.122,-51.271,-179.058,6.192,148.839
C09765=1174.781,92.371,-51.289,-179.056,6.193,148.838
C09766=1174.777,92.621,-51.307,-179.053,6.195,148.838
C09767=1174.772,92.870,-51.325,-179.050,6.195,148.837
C09768=1174.767,93.119,-51.343,-179.047,6.197,148.837
C09769=1174.762,93.368,-51.361,-179.045,6.198,148.836
C09770=1174.757,93.617,-51.379,-179.042,6.199,148.836
C09771=1174.752,93.866,-51.397,-179.040,6.200,148.835
C09772=1174.748,94.116,-51.415,-179.037,6.201,148.835
C09773=1174.743,94.365,-51.433,-179.034,6.203,148.834
C09774=1174.738,94.615,-51.451,-179.032,6.204,148.834
C09775=1174.733,94.864,-51.469,-179.029,6.205,148.833
C09776=1174.728,95.113,-51.487,-179.027,6.206,148.833
C09777=1174.724,95.362,-51.505,-179.024,6.208,148.832
C09778=1174.718,95.612,-51.524,-179.021,6.208,148.832
C09779=1174.713,95.861,-51.542,-179.019,6.210,148.831
C09780=1174.708,96.110,-51.560,-179.015,6.211,148.831
C09781=1174.704,96.360,-51.578,-179.013,6.212,148.830
C09782=1174.699,96.609,-51.596,-179.010,6.214,148.830
C09783=1174.694,96.858,-51.614,-179.008,6.215,148.829
C09784=1174.689,97.107,-51.632,-179.005,6.216,148.829
C09785=1174.684,97.357,-51.650,-179.002,6.218,148.828
C09786=1174.680,97.607,-51.668,-179.000,6.219,148.828
C09787=1174.674,97.856,-51.687,-178.997,6.220,148.827
C09788=1174.670,98.105,-51.706,-178.994,6.221,148.827
C09789=1174.665,98.354,-51.724,-178.992,6.223,148.826
C09790=1174.660,98.603,-51.742,-178.989,6.224,148.826
C09791=1174.655,98.853,-51.760,-178.986,6.225,148.825
C09792=1174.651,99.102,-51.778,-178.984,6.227,148.825
C09793=1174.645,99.351,-51.796,-178.982,6.227,148.824
C09794=1174.640,99.600,-51.815,-178.978,6.229,148.824
C09795=1174.635,99.849,-51.833,-178.976,6.231,148.823
C09796=1174.631,100.099,-51.851,-178.973,6.231,148.823
C09797=1174.626,100.348,-51.869,-178.970,6.233,148.822
C09798=1174.620,100.598,-51.888,-178.968,6.234,148.822
C09799=1174.616,100.846,-51.907,-178.965,6.235,148.821
C09800=1174.612,101.096,-51.925,-178.962,6.237,148.821
C09801=1174.607,101.345,-51.943,-178.960,6.238,148.820
C09802=1174.601,101.595,-51.962,-178.957,6.239,148.820
C09803=1174.597,101.844,-51.981,-178.955,6.240,148.819
C09804=1174.592,102.093,-51.999,-178.952,6.242,148.819
C09805=1174.587,102.342,-52.017,-178.949,6.243,148.818
C09806=1174.582,102.591,-52.036,-178.947,6.244,148.818
C09807=1174.578,102.841,-52.054,-178.944,6.246,148.817
C09808=1174.573,103.090,-52.072,-178.941,6.247,148.817
C09809=1174.567,103.339,-52.092,-178.939,6.248,148.816
C09810=1174.563,103.589,-52.110,-178.936,6.250,148.816
C09811=1174.558,103.838,-52.128,-178.933,6.251,148.815
C09812=1174.553,104.087,-52.147,-178.931,6.252,148.815
C09813=1174.548,104.336,-52.165,-178.928,6.254,148.814
C09814=1174.543,104.586,-52.183,-178.925,6.254,148.814
C09815=1174.539,104.835,-52.202,-178.923,6.256,148.813
C09816=1174.533,105.084,-52.221,-178.920,6.258,148.813
C09817=1174.529,105.334,-52.240,-178.917,6.258,148.812
C09818=1174.524,105.583,-52.258,-178.915,6.260,148.812
C09819=1174.519,105.832,-52.277,-178.912,6.262,148.812
C09820=1174.514,106.101,-52.297,-178.909,6.262,148.811
C09821=1174.509,106.369,-52.317,-178.907,6.264,148.810
C09822=1174.503,106.637,-52.338,-178.903,6.265,148.810
C09823=1174.499,106.906,-52.357,-178.901,6.267,148.809
C09824=1174.494,107.155,-52.375,-178.897,6.268,148.809
C09825=1174.488,107.404,-52.395,-178.895,6.269,148.808
C09826=1174.484,107.654,-52.413,-178.893,6.271,148.808
C09827=1174.479,107.903,-52.432,-178.889,6.272,148.807
C09828=1174.474,108.151,-52.451,-178.887,6.273,148.807
C09829=1174.469,108.402,-52.470,-178.885,6.275,148.807
C09830=1174.464,108.650,-52.489,-178.881,6.276,148.806
C09831=1174.460,108.900,-52.507,-178.879,6.277,148.805
C09832=1174.455,109.149,-52.526,-178.876,6.279,148.805
C09833=1174.450,109.398,-52.544,-178.874,6.281,148.805
C09834=1174.445,109.648,-52.564,-178.871,6.281,148.804
C09835=1174.441,109.896,-52.583,-178.868,6.283,148.804
C09836=1174.436,110.146,-52.602,-178.866,6.285,148.803
C09837=1174.431,110.395,-52.620,-178.863,6.285,148.803
C09838=1174.426,110.645,-52.639,-178.860,6.287,148.802
C09839=1174.421,110.894,-52.658,-178.858,6.289,148.802
C09840=1174.416,111.142,-52.677,-178.855,6.289,148.801
C09841=1174.412,111.392,-52.695,-178.852,6.291,148.801
C09842=1174.406,111.641,-52.715,-178.850,6.293,148.800
C09843=1174.402,111.890,-52.734,-178.848,6.294,148.800
C09844=1174.397,112.140,-52.752,-178.844,6.295,148.799
C09845=1174.392,112.390,-52.772,-178.842,6.297,148.799
C09846=1174.387,112.638,-52.791,-178.839,6.298,148.798
C09847=1174.382,112.888,-52.810,-178.836,6.299,148.798
C09848=1174.378,113.137,-52.828,-178.834,6.301,148.797
C09849=1174.373,113.386,-52.848,-178.831,6.302,148.797
C09850=1174.368,113.635,-52.867,-178.829,6.303,148.797
C09851=1174.363,113.885,-52.886,-178.826,6.305,148.796
C09852=1174.358,114.134,-52.905,-178.823,6.306,148.796
C09853=1174.353,114.383,-52.924,-178.821,6.307,148.795
C09854=1174.348,114.632,-52.943,-178.818,6.309,148.795
C09855=1174.343,114.881,-52.963,-178.815,6.310,148.794
C09856=1174.339,115.130,-52.982,-178.812,6.312,148.794
C09857=1174.334,115.380,-53.001,-178.810,6.313,148.793
C09858=1174.329,115.629,-53.019,-178.807,6.315,148.793
C09859=1174.325,115.879,-53.039,-178.804,6.316,148.792
C09860=1174.319,116.127,-53.058,-178.802,6.317,148.792
C09861=1174.315,116.377,-53.077,-178.799,6.319,148.791
C09862=1174.310,116.626,-53.097,-178.796,6.320,148.791
C09863=1174.305,116.875,-53.116,-178.793,6.322,148.790
C09864=1174.301,117.124,-53.135,-178.791,6.323,148.790
C09865=1174.296,117.374,-53.154,-178.788,6.324,148.789
C09866=1174.290,117.623,-53.173,-178.785,6.326,148.789
C09867=1174.286,117.872,-53.193,-178.783,6.327,148.789
C09868=1174.281,118.121,-53.212,-178.780,6.329,148.788
C09869=1174.276,118.370,-53.231,-178.777,6.330,148.788
C09870=1174.271,118.620,-53.251,-178.775,6.332,148.787
C09871=1174.267,118.869,-53.270,-178.772,6.333,148.787
C09872=1174.262,119.118,-53.289,-178.770,6.334,148.786
C09873=1174.257,119.367,-53.309,-178.767,6.336,148.786
C09874=1174.252,119.617,-53.328,-178.764,6.338,148.785
C09875=1174.248,119.866,-53.347,-178.762,6.338,148.785
C09876=1174.243,120.115,-53.367,-178.759,6.340,148.785
C09877=1174.238,120.364,-53.386,-178.756,6.342,148.784
C09878=1174.233,120.613,-53.405,-178.753,6.343,148.783
C09879=1174.228,120.863,-53.425,-178.751,6.344,148.783
C09880=1174.224,121.112,-53.444,-178.748,6.346,148.783
C09881=1174.219,121.361,-53.463,-178.745,6.347,148.782
C09882=1174.214,121.610,-53.484,-178.742,6.349,148.782
C09883=1174.209,121.859,-53.503,-178.740,6.350,148.781
C09884=1174.204,122.108,-53.523,-178.738,6.352,148.781
C09885=1174.200,122.357,-53.542,-178.734,6.353,148.780
C09886=1174.195,122.606,-53.561,-178.732,6.355,148.780
C09887=1174.190,122.856,-53.581,-178.730,6.356,148.779
C09888=1174.185,123.105,-53.600,-178.727,6.357,148.779
C09889=1174.180,123.354,-53.620,-178.724,6.359,148.779
C09890=1174.175,123.603,-53.640,-178.721,6.361,148.778
C09891=1174.171,123.853,-53.660,-178.719,6.361,148.778
C09892=1174.166,124.101,-53.678,-178.716,6.363,148.777
C09893=1174.161,124.351,-53.698,-178.713,6.365,148.777
C09894=1174.157,124.601,-53.718,-178.710,6.366,148.776
C09895=1174.152,124.849,-53.738,-178.707,6.368,148.776
C09896=1174.147,125.098,-53.757,-178.705,6.369,148.775
C09897=1174.142,125.348,-53.777,-178.703,6.371,148.775
C09898=1174.137,125.597,-53.797,-178.700,6.372,148.775
C09899=1174.132,125.846,-53.817,-178.697,6.374,148.774
C09900=1174.127,126.095,-53.836,-178.695,6.375,148.774
C09901=1174.123,126.345,-53.856,-178.692,6.376,148.773
C09902=1174.117,126.594,-53.875,-178.689,6.378,148.773
C09903=1174.113,126.843,-53.896,-178.687,6.380,148.772
C09904=1174.108,127.092,-53.915,-178.683,6.381,148.772
C09905=1174.103,127.342,-53.935,-178.681,6.382,148.771
C09906=1174.099,127.590,-53.954,-178.678,6.384,148.771
C09907=1174.094,127.839,-53.974,-178.676,6.386,148.771
C09908=1174.090,128.088,-53.994,-178.673,6.387,148.770
C09909=1174.085,128.338,-54.014,-178.670,6.389,148.770
C09910=1174.080,128.587,-54.033,-178.668,6.390,148.769
C09911=1174.075,128.836,-54.054,-178.665,6.392,148.769
C09912=1174.070,129.086,-54.074,-178.662,6.393,148.768
C09913=1174.065,129.335,-54.094,-178.660,6.395,148.768
C09914=1174.060,129.583,-54.114,-178.656,6.396,148.767
C09915=1174.055,129.833,-54.133,-178.654,6.397,148.767
C09916=1174.051,130.082,-54.154,-178.652,6.399,148.767
C09917=1174.046,130.331,-54.173,-178.649,6.401,148.766
C09918=1174.042,130.580,-54.194,-178.646,6.403,148.766
C09919=1174.037,130.829,-54.213,-178.643,6.404,148.765
C09920=1174.032,131.078,-54.233,-178.640,6.406,148.765
C09921=1174.027,131.328,-54.253,-178.638,6.407,148.764
C09922=1174.023,131.577,-54.273,-178.636,6.408,148.764
C09923=1174.018,131.826,-54.293,-178.633,6.410,148.764
C09924=1174.013,132.095,-54.316,-178.630,6.411,148.763
C09925=1174.008,132.363,-54.337,-178.627,6.413,148.763
C09926=1174.002,132.632,-54.358,-178.624,6.415,148.762
C09927=1173.998,132.900,-54.380,-178.621,6.416,148.762
C09928=1173.992,133.149,-54.399,-178.618,6.418,148.761
C09929=1173.987,133.398,-54.420,-178.616,6.420,148.761
C09930=1173.982,133.648,-54.440,-178.613,6.422,148.760
C09931=1173.978,133.897,-54.460,-178.610,6.423,148.760
C09932=1173.973,134.146,-54.481,-178.608,6.424,148.760
C09933=1173.969,134.395,-54.500,-178.605,6.426,148.759
C09934=1173.964,134.644,-54.521,-178.602,6.427,148.759
C09935=1173.959,134.894,-54.541,-178.600,6.429,148.758
C09936=1173.954,135.143,-54.561,-178.597,6.431,148.758
C09937=1173.949,135.391,-54.581,-178.594,6.433,148.757
C09938=1173.945,135.641,-54.601,-178.592,6.433,148.757
C09939=1173.940,135.890,-54.621,-178.589,6.435,148.756
C09940=1173.935,136.139,-54.642,-178.586,6.437,148.756
C09941=1173.931,136.388,-54.663,-178.583,6.438,148.756
C09942=1173.926,136.638,-54.682,-178.581,6.440,148.755
C09943=1173.921,136.887,-54.703,-178.578,6.442,148.755
C09944=1173.916,137.136,-54.724,-178.575,6.444,148.754
C09945=1173.911,137.384,-54.744,-178.573,6.444,148.754
C09946=1173.906,137.634,-54.763,-178.570,6.446,148.753
C09947=1173.901,137.883,-54.784,-178.567,6.448,148.753
C09948=1173.897,138.132,-54.805,-178.565,6.449,148.753
C09949=1173.892,138.381,-54.825,-178.562,6.451,148.752
C09950=1173.888,138.630,-54.846,-178.559,6.453,148.752
C09951=1173.882,138.880,-54.866,-178.557,6.455,148.752
C09952=1173.878,139.129,-54.886,-178.554,6.456,148.751
C09953=1173.874,139.378,-54.907,-178.551,6.457,148.750
C09954=1173.868,139.627,-54.927,-178.549,6.459,148.750
C09955=1173.864,139.876,-54.948,-178.546,6.460,148.750
C09956=1173.860,140.125,-54.968,-178.543,6.462,148.749
C09957=1173.854,140.375,-54.988,-178.540,6.464,148.749
C09958=1173.850,140.624,-55.009,-178.538,6.466,148.749
C09959=1173.845,140.873,-55.029,-178.535,6.467,148.748
C09960=1173.840,141.122,-55.050,-178.532,6.469,148.748
C09961=1173.836,141.371,-55.071,-178.530,6.470,148.747
C09962=1173.830,141.620,-55.092,-178.527,6.471,148.747
C09963=1173.826,141.869,-55.112,-178.524,6.473,148.746
C09964=1173.822,142.118,-55.132,-178.522,6.475,148.746
C09965=1173.816,142.367,-55.153,-178.519,6.477,148.746
C09966=1173.812,142.616,-55.174,-178.516,6.478,148.745
C09967=1173.807,142.865,-55.195,-178.514,6.480,148.745
C09968=1173.802,143.114,-55.215,-178.511,6.482,148.744
C09969=1173.798,143.363,-55.235,-178.508,6.484,148.744
C09970=1173.793,143.613,-55.256,-178.506,6.485,148.744
C09971=1173.788,143.862,-55.277,-178.503,6.486,148.743
C09972=1173.783,144.111,-55.298,-178.500,6.488,148.743
C09973=1173.779,144.360,-55.318,-178.498,6.490,148.742
C09974=1173.773,144.609,-55.339,-178.495,6.491,148.742
C09975=1173.769,144.858,-55.359,-178.492,6.493,148.742
C09976=1173.764,145.107,-55.380,-178.489,6.495,148.741
C09977=1173.760,145.356,-55.402,-178.487,6.497,148.741
C09978=1173.755,145.605,-55.423,-178.484,6.498,148.740
C09979=1173.751,145.854,-55.443,-178.481,6.500,148.740
C09980=1173.746,146.104,-55.464,-178.479,6.502,148.740
C09981=1173.741,146.353,-55.484,-178.476,6.504,148.739
C09982=1173.736,146.602,-55.505,-178.473,6.505,148.739
C09983=1173.731,146.851,-55.526,-178.471,6.506,148.738
C09984=1173.727,147.099,-55.547,-178.468,6.508,148.738
C09985=1173.721,147.349,-55.568,-178.465,6.509,148.737
C09986=1173.717,147.598,-55.589,-178.463,6.511,148.737
C09987=1173.712,147.847,-55.610,-178.460,6.513,148.737
C09988=1173.708,148.097,-55.630,-178.457,6.515,148.736
C09989=1173.703,148.345,-55.652,-178.454,6.516,148.736
C09990=1173.699,148.594,-55.673,-178.452,6.518,148.736
C09991=1173.694,148.843,-55.694,-178.449,6.520,148.735
C09992=1173.688,149.093,-55.714,-178.446,6.522,148.735
C09993=1173.684,149.341,-55.736,-178.444,6.523,148.734
C09994=1173.679,149.590,-55.757,-178.441,6.525,148.734
C09995=1173.674,149.840,-55.778,-178.438,6.527,148.734
C09996=1173.670,150.089,-55.798,-178.435,6.528,148.733
//INST
///DATE 2021/06/25 14:29
///ATTR SC,RW,RJ
////FRAME ROBOT
///GROUP1 RB1
NOP
MOVL C00000 V=800.0 PL=0
MOVL C00001 V=800.0 PL=0
MOVL C00002 V=800.0 PL=0
MOVL C00003 V=800.0 PL=0
MOVL C00004 V=800.0 PL=0
MOVL C00005 V=800.0 PL=0
MOVL C00006 V=800.0 PL=0
MOVL C00007 V=800.0 PL=0
MOVL C00008 V=800.0 PL=0
MOVL C00009 V=800.0 PL=0
MOVL C00010 V=800.0 PL=0
MOVL C00011 V=800.0 PL=0
MOVL C00012 V=800.0 PL=0
MOVL C00013 V=800.0 PL=0
MOVL C00014 V=800.0 PL=0
MOVL C00015 V=800.0 PL=0
MOVL C00016 V=800.0 PL=0
MOVL C00017 V=800.0 PL=0
MOVL C00018 V=800.0 PL=0
MOVL C00019 V=800.0 PL=0
MOVL C00020 V=800.0 PL=0
MOVL C00021 V=800.0 PL=0
MOVL C00022 V=800.0 PL=0
MOVL C00023 V=800.0 PL=0
MOVL C00024 V=800.0 PL=0
MOVL C00025 V=800.0 PL=0
MOVL C00026 V=800.0 PL=0
MOVL C00027 V=800.0 PL=0
MOVL C00028 V=800.0 PL=0
MOVL C00029 V=800.0 PL=0
MOVL C00030 V=800.0 PL=0
MOVL C00031 V=800.0 PL=0
MOVL C00032 V=800.0 PL=0
MOVL C00033 V=800.0 PL=0
MOVL C00034 V=800.0 PL=0
MOVL C00035 V=800.0 PL=0
MOVL C00036 V=800.0 PL=0
MOVL C00037 V=800.0 PL=0
MOVL C00038 V=800.0 PL=0
MOVL C00039 V=800.0 PL=0
MOVL C00040 V=800.0 PL=0
MOVL C00041 V=800.0 PL=0
MOVL C00042 V=800.0 PL=0
MOVL C00043 V=800.0 PL=0
MOVL C00044 V=800.0 PL=0
MOVL C00045 V=800.0 PL=0
MOVL C00046 V=800.0 PL=0
MOVL C00047 V=800.0 PL=0
MOVL C00048 V=800.0 PL=0
MOVL C00049 V=800.0 PL=0
MOVL C00050 V=800.0 PL=0
MOVL C00051 V=800.0 PL=0
MOVL C00052 V=800.0 PL=0
MOVL C00053 V=800.0 PL=0
MOVL C00054 V=800.0 PL=0
MOVL C00055 V=800.0 PL=0
MOVL C00056 V=800.0 PL=0
MOVL C00057 V=800.0 PL=0
MOVL C00058 V=800.0 PL=0
MOVL C00059 V=800.0 PL=0
MOVL C00060 V=800.0 PL=0
MOVL C00061 V=800.0 PL=0
MOVL C00062 V=800.0 PL=0
MOVL C00063 V=800.0 PL=0
MOVL C00064 V=800.0 PL=0
MOVL C00065 V=800.0 PL=0
MOVL C00066 V=800.0 PL=0
MOVL C00067 V=800.0 PL=0
MOVL C00068 V=800.0 PL=0
MOVL C00069 V=800.0 PL=0
MOVL C00070 V=800.0 PL=0
MOVL C00071 V=800.0 PL=0
MOVL C00072 V=800.0 PL=0
MOVL C00073 V=800.0 PL=0
MOVL C00074 V=800.0 PL=0
MOVL C00075 V=800.0 PL=0
MOVL C00076 V=800.0 PL=0
MOVL C00077 V=800.0 PL=0
MOVL C00078 V=800.0 PL=0
MOVL C00079 V=800.0 PL=0
MOVL C00080 V=800.0 PL=0
MOVL C00081 V=800.0 PL=0
MOVL C00082 V=800.0 PL=0
MOVL C00083 V=800.0 PL=0
MOVL C00084 V=800.0 PL=0
MOVL C00085 V=800.0 PL=0
MOVL C00086 V=800.0 PL=0
MOVL C00087 V=800.0 PL=0
MOVL C00088 V=800.0 PL=0
MOVL C00089 V=800.0 PL=0
MOVL C00090 V=800.0 PL=0
MOVL C00091 V=800.0 PL=0
MOVL C00092 V=800.0 PL=0
MOVL C00093 V=800.0 PL=0
MOVL C00094 V=800.0 PL=0
MOVL C00095 V=800.0 PL=0
MOVL C00096 V=800.0 PL=0
MOVL C00097 V=800.0 PL=0
MOVL C00098 V=800.0 PL=0
MOVL C00099 V=800.0 PL=0
MOVL C00100 V=800.0 PL=0
MOVL C00101 V=800.0 PL=0
MOVL C00102 V=800.0 PL=0
MOVL C00103 V=800.0 PL=0
MOVL C00104 V=800.0 PL=0
MOVL C00105 V=800.0 PL=0
MOVL C00106 V=800.0 PL=0
MOVL C00107 V=800.0 PL=0
MOVL C00108 V=800.0 PL=0
MOVL C00109 V=800.0 PL=0
MOVL C00110 V=800.0 PL=0
MOVL C00111 V=800.0 PL=0
MOVL C00112 V=800.0 PL=0
MOVL C00113 V=800.0 PL=0
MOVL C00114 V=800.0 PL=0
MOVL C00115 V=800.0 PL=0
MOVL C00116 V=800.0 PL=0
MOVL C00117 V=800.0 PL=0
MOVL C00118 V=800.0 PL=0
MOVL C00119 V=800.0 PL=0
MOVL C00120 V=800.0 PL=0
MOVL C00121 V=800.0 PL=0
MOVL C00122 V=800.0 PL=0
MOVL C00123 V=800.0 PL=0
MOVL C00124 V=800.0 PL=0
MOVL C00125 V=800.0 PL=0
MOVL C00126 V=800.0 PL=0
MOVL C00127 V=800.0 PL=0
MOVL C00128 V=800.0 PL=0
MOVL C00129 V=800.0 PL=0
MOVL C00130 V=800.0 PL=0
MOVL C00131 V=800.0 PL=0
MOVL C00132 V=800.0 PL=0
MOVL C00133 V=800.0 PL=0
MOVL C00134 V=800.0 PL=0
MOVL C00135 V=800.0 PL=0
MOVL C00136 V=800.0 PL=0
MOVL C00137 V=800.0 PL=0
MOVL C00138 V=800.0 PL=0
MOVL C00139 V=800.0 PL=0
MOVL C00140 V=800.0 PL=0
MOVL C00141 V=800.0 PL=0
MOVL C00142 V=800.0 PL=0
MOVL C00143 V=800.0 PL=0
MOVL C00144 V=800.0 PL=0
MOVL C00145 V=800.0 PL=0
MOVL C00146 V=800.0 PL=0
MOVL C00147 V=800.0 PL=0
MOVL C00148 V=800.0 PL=0
MOVL C00149 V=800.0 PL=0
MOVL C00150 V=800.0 PL=0
MOVL C00151 V=800.0 PL=0
MOVL C00152 V=800.0 PL=0
MOVL C00153 V=800.0 PL=0
MOVL C00154 V=800.0 PL=0
MOVL C00155 V=800.0 PL=0
MOVL C00156 V=800.0 PL=0
MOVL C00157 V=800.0 PL=0
MOVL C00158 V=800.0 PL=0
MOVL C00159 V=800.0 PL=0
MOVL C00160 V=800.0 PL=0
MOVL C00161 V=800.0 PL=0
MOVL C00162 V=800.0 PL=0
MOVL C00163 V=800.0 PL=0
MOVL C00164 V=800.0 PL=0
MOVL C00165 V=800.0 PL=0
MOVL C00166 V=800.0 PL=0
MOVL C00167 V=800.0 PL=0
MOVL C00168 V=800.0 PL=0
MOVL C00169 V=800.0 PL=0
MOVL C00170 V=800.0 PL=0
MOVL C00171 V=800.0 PL=0
MOVL C00172 V=800.0 PL=0
MOVL C00173 V=800.0 PL=0
MOVL C00174 V=800.0 PL=0
MOVL C00175 V=800.0 PL=0
MOVL C00176 V=800.0 PL=0
MOVL C00177 V=800.0 PL=0
MOVL C00178 V=800.0 PL=0
MOVL C00179 V=800.0 PL=0
MOVL C00180 V=800.0 PL=0
MOVL C00181 V=800.0 PL=0
MOVL C00182 V=800.0 PL=0
MOVL C00183 V=800.0 PL=0
MOVL C00184 V=800.0 PL=0
MOVL C00185 V=800.0 PL=0
MOVL C00186 V=800.0 PL=0
MOVL C00187 V=800.0 PL=0
MOVL C00188 V=800.0 PL=0
MOVL C00189 V=800.0 PL=0
MOVL C00190 V=800.0 PL=0
MOVL C00191 V=800.0 PL=0
MOVL C00192 V=800.0 PL=0
MOVL C00193 V=800.0 PL=0
MOVL C00194 V=800.0 PL=0
MOVL C00195 V=800.0 PL=0
MOVL C00196 V=800.0 PL=0
MOVL C00197 V=800.0 PL=0
MOVL C00198 V=800.0 PL=0
MOVL C00199 V=800.0 PL=0
MOVL C00200 V=800.0 PL=0
MOVL C00201 V=800.0 PL=0
MOVL C00202 V=800.0 PL=0
MOVL C00203 V=800.0 PL=0
MOVL C00204 V=800.0 PL=0
MOVL C00205 V=800.0 PL=0
MOVL C00206 V=800.0 PL=0
MOVL C00207 V=800.0 PL=0
MOVL C00208 V=800.0 PL=0
MOVL C00209 V=800.0 PL=0
MOVL C00210 V=800.0 PL=0
MOVL C00211 V=800.0 PL=0
MOVL C00212 V=800.0 PL=0
MOVL C00213 V=800.0 PL=0
MOVL C00214 V=800.0 PL=0
MOVL C00215 V=800.0 PL=0
MOVL C00216 V=800.0 PL=0
MOVL C00217 V=800.0 PL=0
MOVL C00218 V=800.0 PL=0
MOVL C00219 V=800.0 PL=0
MOVL C00220 V=800.0 PL=0
MOVL C00221 V=800.0 PL=0
MOVL C00222 V=800.0 PL=0
MOVL C00223 V=800.0 PL=0
MOVL C00224 V=800.0 PL=0
MOVL C00225 V=800.0 PL=0
MOVL C00226 V=800.0 PL=0
MOVL C00227 V=800.0 PL=0
MOVL C00228 V=800.0 PL=0
MOVL C00229 V=800.0 PL=0
MOVL C00230 V=800.0 PL=0
MOVL C00231 V=800.0 PL=0
MOVL C00232 V=800.0 PL=0
MOVL C00233 V=800.0 PL=0
MOVL C00234 V=800.0 PL=0
MOVL C00235 V=800.0 PL=0
MOVL C00236 V=800.0 PL=0
MOVL C00237 V=800.0 PL=0
MOVL C00238 V=800.0 PL=0
MOVL C00239 V=800.0 PL=0
MOVL C00240 V=800.0 PL=0
MOVL C00241 V=800.0 PL=0
MOVL C00242 V=800.0 PL=0
MOVL C00243 V=800.0 PL=0
MOVL C00244 V=800.0 PL=0
MOVL C00245 V=800.0 PL=0
MOVL C00246 V=800.0 PL=0
MOVL C00247 V=800.0 PL=0
MOVL C00248 V=800.0 PL=0
MOVL C00249 V=800.0 PL=0
MOVL C00250 V=800.0 PL=0
MOVL C00251 V=800.0 PL=0
MOVL C00252 V=800.0 PL=0
MOVL C00253 V=800.0 PL=0
MOVL C00254 V=800.0 PL=0
MOVL C00255 V=800.0 PL=0
MOVL C00256 V=800.0 PL=0
MOVL C00257 V=800.0 PL=0
MOVL C00258 V=800.0 PL=0
MOVL C00259 V=800.0 PL=0
MOVL C00260 V=800.0 PL=0
MOVL C00261 V=800.0 PL=0
MOVL C00262 V=800.0 PL=0
MOVL C00263 V=800.0 PL=0
MOVL C00264 V=800.0 PL=0
MOVL C00265 V=800.0 PL=0
MOVL C00266 V=800.0 PL=0
MOVL C00267 V=800.0 PL=0
MOVL C00268 V=800.0 PL=0
MOVL C00269 V=800.0 PL=0
MOVL C00270 V=800.0 PL=0
MOVL C00271 V=800.0 PL=0
MOVL C00272 V=800.0 PL=0
MOVL C00273 V=800.0 PL=0
MOVL C00274 V=800.0 PL=0
MOVL C00275 V=800.0 PL=0
MOVL C00276 V=800.0 PL=0
MOVL C00277 V=800.0 PL=0
MOVL C00278 V=800.0 PL=0
MOVL C00279 V=800.0 PL=0
MOVL C00280 V=800.0 PL=0
MOVL C00281 V=800.0 PL=0
MOVL C00282 V=800.0 PL=0
MOVL C00283 V=800.0 PL=0
MOVL C00284 V=800.0 PL=0
MOVL C00285 V=800.0 PL=0
MOVL C00286 V=800.0 PL=0
MOVL C00287 V=800.0 PL=0
MOVL C00288 V=800.0 PL=0
MOVL C00289 V=800.0 PL=0
MOVL C00290 V=800.0 PL=0
MOVL C00291 V=800.0 PL=0
MOVL C00292 V=800.0 PL=0
MOVL C00293 V=800.0 PL=0
MOVL C00294 V=800.0 PL=0
MOVL C00295 V=800.0 PL=0
MOVL C00296 V=800.0 PL=0
MOVL C00297 V=800.0 PL=0
MOVL C00298 V=800.0 PL=0
MOVL C00299 V=800.0 PL=0
MOVL C00300 V=800.0 PL=0
MOVL C00301 V=800.0 PL=0
MOVL C00302 V=800.0 PL=0
MOVL C00303 V=800.0 PL=0
MOVL C00304 V=800.0 PL=0
MOVL C00305 V=800.0 PL=0
MOVL C00306 V=800.0 PL=0
MOVL C00307 V=800.0 PL=0
MOVL C00308 V=800.0 PL=0
MOVL C00309 V=800.0 PL=0
MOVL C00310 V=800.0 PL=0
MOVL C00311 V=800.0 PL=0
MOVL C00312 V=800.0 PL=0
MOVL C00313 V=800.0 PL=0
MOVL C00314 V=800.0 PL=0
MOVL C00315 V=800.0 PL=0
MOVL C00316 V=800.0 PL=0
MOVL C00317 V=800.0 PL=0
MOVL C00318 V=800.0 PL=0
MOVL C00319 V=800.0 PL=0
MOVL C00320 V=800.0 PL=0
MOVL C00321 V=800.0 PL=0
MOVL C00322 V=800.0 PL=0
MOVL C00323 V=800.0 PL=0
MOVL C00324 V=800.0 PL=0
MOVL C00325 V=800.0 PL=0
MOVL C00326 V=800.0 PL=0
MOVL C00327 V=800.0 PL=0
MOVL C00328 V=800.0 PL=0
MOVL C00329 V=800.0 PL=0
MOVL C00330 V=800.0 PL=0
MOVL C00331 V=800.0 PL=0
MOVL C00332 V=800.0 PL=0
MOVL C00333 V=800.0 PL=0
MOVL C00334 V=800.0 PL=0
MOVL C00335 V=800.0 PL=0
MOVL C00336 V=800.0 PL=0
MOVL C00337 V=800.0 PL=0
MOVL C00338 V=800.0 PL=0
MOVL C00339 V=800.0 PL=0
MOVL C00340 V=800.0 PL=0
MOVL C00341 V=800.0 PL=0
MOVL C00342 V=800.0 PL=0
MOVL C00343 V=800.0 PL=0
MOVL C00344 V=800.0 PL=0
MOVL C00345 V=800.0 PL=0
MOVL C00346 V=800.0 PL=0
MOVL C00347 V=800.0 PL=0
MOVL C00348 V=800.0 PL=0
MOVL C00349 V=800.0 PL=0
MOVL C00350 V=800.0 PL=0
MOVL C00351 V=800.0 PL=0
MOVL C00352 V=800.0 PL=0
MOVL C00353 V=800.0 PL=0
MOVL C00354 V=800.0 PL=0
MOVL C00355 V=800.0 PL=0
MOVL C00356 V=800.0 PL=0
MOVL C00357 V=800.0 PL=0
MOVL C00358 V=800.0 PL=0
MOVL C00359 V=800.0 PL=0
MOVL C00360 V=800.0 PL=0
MOVL C00361 V=800.0 PL=0
MOVL C00362 V=800.0 PL=0
MOVL C00363 V=800.0 PL=0
MOVL C00364 V=800.0 PL=0
MOVL C00365 V=800.0 PL=0
MOVL C00366 V=800.0 PL=0
MOVL C00367 V=800.0 PL=0
MOVL C00368 V=800.0 PL=0
MOVL C00369 V=800.0 PL=0
MOVL C00370 V=800.0 PL=0
MOVL C00371 V=800.0 PL=0
MOVL C00372 V=800.0 PL=0
MOVL C00373 V=800.0 PL=0
MOVL C00374 V=800.0 PL=0
MOVL C00375 V=800.0 PL=0
MOVL C00376 V=800.0 PL=0
MOVL C00377 V=800.0 PL=0
MOVL C00378 V=800.0 PL=0
MOVL C00379 V=800.0 PL=0
MOVL C00380 V=800.0 PL=0
MOVL C00381 V=800.0 PL=0
MOVL C00382 V=800.0 PL=0
MOVL C00383 V=800.0 PL=0
MOVL C00384 V=800.0 PL=0
MOVL C00385 V=800.0 PL=0
MOVL C00386 V=800.0 PL=0
MOVL C00387 V=800.0 PL=0
MOVL C00388 V=800.0 PL=0
MOVL C00389 V=800.0 PL=0
MOVL C00390 V=800.0 PL=0
MOVL C00391 V=800.0 PL=0
MOVL C00392 V=800.0 PL=0
MOVL C00393 V=800.0 PL=0
MOVL C00394 V=800.0 PL=0
MOVL C00395 V=800.0 PL=0
MOVL C00396 V=800.0 PL=0
MOVL C00397 V=800.0 PL=0
MOVL C00398 V=800.0 PL=0
MOVL C00399 V=800.0 PL=0
MOVL C00400 V=800.0 PL=0
MOVL C00401 V=800.0 PL=0
MOVL C00402 V=800.0 PL=0
MOVL C00403 V=800.0 PL=0
MOVL C00404 V=800.0 PL=0
MOVL C00405 V=800.0 PL=0
MOVL C00406 V=800.0 PL=0
MOVL C00407 V=800.0 PL=0
MOVL C00408 V=800.0 PL=0
MOVL C00409 V=800.0 PL=0
MOVL C00410 V=800.0 PL=0
MOVL C00411 V=800.0 PL=0
MOVL C00412 V=800.0 PL=0
MOVL C00413 V=800.0 PL=0
MOVL C00414 V=800.0 PL=0
MOVL C00415 V=800.0 PL=0
MOVL C00416 V=800.0 PL=0
MOVL C00417 V=800.0 PL=0
MOVL C00418 V=800.0 PL=0
MOVL C00419 V=800.0 PL=0
MOVL C00420 V=800.0 PL=0
MOVL C00421 V=800.0 PL=0
MOVL C00422 V=800.0 PL=0
MOVL C00423 V=800.0 PL=0
MOVL C00424 V=800.0 PL=0
MOVL C00425 V=800.0 PL=0
MOVL C00426 V=800.0 PL=0
MOVL C00427 V=800.0 PL=0
MOVL C00428 V=800.0 PL=0
MOVL C00429 V=800.0 PL=0
MOVL C00430 V=800.0 PL=0
MOVL C00431 V=800.0 PL=0
MOVL C00432 V=800.0 PL=0
MOVL C00433 V=800.0 PL=0
MOVL C00434 V=800.0 PL=0
MOVL C00435 V=800.0 PL=0
MOVL C00436 V=800.0 PL=0
MOVL C00437 V=800.0 PL=0
MOVL C00438 V=800.0 PL=0
MOVL C00439 V=800.0 PL=0
MOVL C00440 V=800.0 PL=0
MOVL C00441 V=800.0 PL=0
MOVL C00442 V=800.0 PL=0
MOVL C00443 V=800.0 PL=0
MOVL C00444 V=800.0 PL=0
MOVL C00445 V=800.0 PL=0
MOVL C00446 V=800.0 PL=0
MOVL C00447 V=800.0 PL=0
MOVL C00448 V=800.0 PL=0
MOVL C00449 V=800.0 PL=0
MOVL C00450 V=800.0 PL=0
MOVL C00451 V=800.0 PL=0
MOVL C00452 V=800.0 PL=0
MOVL C00453 V=800.0 PL=0
MOVL C00454 V=800.0 PL=0
MOVL C00455 V=800.0 PL=0
MOVL C00456 V=800.0 PL=0
MOVL C00457 V=800.0 PL=0
MOVL C00458 V=800.0 PL=0
MOVL C00459 V=800.0 PL=0
MOVL C00460 V=800.0 PL=0
MOVL C00461 V=800.0 PL=0
MOVL C00462 V=800.0 PL=0
MOVL C00463 V=800.0 PL=0
MOVL C00464 V=800.0 PL=0
MOVL C00465 V=800.0 PL=0
MOVL C00466 V=800.0 PL=0
MOVL C00467 V=800.0 PL=0
MOVL C00468 V=800.0 PL=0
MOVL C00469 V=800.0 PL=0
MOVL C00470 V=800.0 PL=0
MOVL C00471 V=800.0 PL=0
MOVL C00472 V=800.0 PL=0
MOVL C00473 V=800.0 PL=0
MOVL C00474 V=800.0 PL=0
MOVL C00475 V=800.0 PL=0
MOVL C00476 V=800.0 PL=0
MOVL C00477 V=800.0 PL=0
MOVL C00478 V=800.0 PL=0
MOVL C00479 V=800.0 PL=0
MOVL C00480 V=800.0 PL=0
MOVL C00481 V=800.0 PL=0
MOVL C00482 V=800.0 PL=0
MOVL C00483 V=800.0 PL=0
MOVL C00484 V=800.0 PL=0
MOVL C00485 V=800.0 PL=0
MOVL C00486 V=800.0 PL=0
MOVL C00487 V=800.0 PL=0
MOVL C00488 V=800.0 PL=0
MOVL C00489 V=800.0 PL=0
MOVL C00490 V=800.0 PL=0
MOVL C00491 V=800.0 PL=0
MOVL C00492 V=800.0 PL=0
MOVL C00493 V=800.0 PL=0
MOVL C00494 V=800.0 PL=0
MOVL C00495 V=800.0 PL=0
MOVL C00496 V=800.0 PL=0
MOVL C00497 V=800.0 PL=0
MOVL C00498 V=800.0 PL=0
MOVL C00499 V=800.0 PL=0
MOVL C00500 V=800.0 PL=0
MOVL C00501 V=800.0 PL=0
MOVL C00502 V=800.0 PL=0
MOVL C00503 V=800.0 PL=0
MOVL C00504 V=800.0 PL=0
MOVL C00505 V=800.0 PL=0
MOVL C00506 V=800.0 PL=0
MOVL C00507 V=800.0 PL=0
MOVL C00508 V=800.0 PL=0
MOVL C00509 V=800.0 PL=0
MOVL C00510 V=800.0 PL=0
MOVL C00511 V=800.0 PL=0
MOVL C00512 V=800.0 PL=0
MOVL C00513 V=800.0 PL=0
MOVL C00514 V=800.0 PL=0
MOVL C00515 V=800.0 PL=0
MOVL C00516 V=800.0 PL=0
MOVL C00517 V=800.0 PL=0
MOVL C00518 V=800.0 PL=0
MOVL C00519 V=800.0 PL=0
MOVL C00520 V=800.0 PL=0
MOVL C00521 V=800.0 PL=0
MOVL C00522 V=800.0 PL=0
MOVL C00523 V=800.0 PL=0
MOVL C00524 V=800.0 PL=0
MOVL C00525 V=800.0 PL=0
MOVL C00526 V=800.0 PL=0
MOVL C00527 V=800.0 PL=0
MOVL C00528 V=800.0 PL=0
MOVL C00529 V=800.0 PL=0
MOVL C00530 V=800.0 PL=0
MOVL C00531 V=800.0 PL=0
MOVL C00532 V=800.0 PL=0
MOVL C00533 V=800.0 PL=0
MOVL C00534 V=800.0 PL=0
MOVL C00535 V=800.0 PL=0
MOVL C00536 V=800.0 PL=0
MOVL C00537 V=800.0 PL=0
MOVL C00538 V=800.0 PL=0
MOVL C00539 V=800.0 PL=0
MOVL C00540 V=800.0 PL=0
MOVL C00541 V=800.0 PL=0
MOVL C00542 V=800.0 PL=0
MOVL C00543 V=800.0 PL=0
MOVL C00544 V=800.0 PL=0
MOVL C00545 V=800.0 PL=0
MOVL C00546 V=800.0 PL=0
MOVL C00547 V=800.0 PL=0
MOVL C00548 V=800.0 PL=0
MOVL C00549 V=800.0 PL=0
MOVL C00550 V=800.0 PL=0
MOVL C00551 V=800.0 PL=0
MOVL C00552 V=800.0 PL=0
MOVL C00553 V=800.0 PL=0
MOVL C00554 V=800.0 PL=0
MOVL C00555 V=800.0 PL=0
MOVL C00556 V=800.0 PL=0
MOVL C00557 V=800.0 PL=0
MOVL C00558 V=800.0 PL=0
MOVL C00559 V=800.0 PL=0
MOVL C00560 V=800.0 PL=0
MOVL C00561 V=800.0 PL=0
MOVL C00562 V=800.0 PL=0
MOVL C00563 V=800.0 PL=0
MOVL C00564 V=800.0 PL=0
MOVL C00565 V=800.0 PL=0
MOVL C00566 V=800.0 PL=0
MOVL C00567 V=800.0 PL=0
MOVL C00568 V=800.0 PL=0
MOVL C00569 V=800.0 PL=0
MOVL C00570 V=800.0 PL=0
MOVL C00571 V=800.0 PL=0
MOVL C00572 V=800.0 PL=0
MOVL C00573 V=800.0 PL=0
MOVL C00574 V=800.0 PL=0
MOVL C00575 V=800.0 PL=0
MOVL C00576 V=800.0 PL=0
MOVL C00577 V=800.0 PL=0
MOVL C00578 V=800.0 PL=0
MOVL C00579 V=800.0 PL=0
MOVL C00580 V=800.0 PL=0
MOVL C00581 V=800.0 PL=0
MOVL C00582 V=800.0 PL=0
MOVL C00583 V=800.0 PL=0
MOVL C00584 V=800.0 PL=0
MOVL C00585 V=800.0 PL=0
MOVL C00586 V=800.0 PL=0
MOVL C00587 V=800.0 PL=0
MOVL C00588 V=800.0 PL=0
MOVL C00589 V=800.0 PL=0
MOVL C00590 V=800.0 PL=0
MOVL C00591 V=800.0 PL=0
MOVL C00592 V=800.0 PL=0
MOVL C00593 V=800.0 PL=0
MOVL C00594 V=800.0 PL=0
MOVL C00595 V=800.0 PL=0
MOVL C00596 V=800.0 PL=0
MOVL C00597 V=800.0 PL=0
MOVL C00598 V=800.0 PL=0
MOVL C00599 V=800.0 PL=0
MOVL C00600 V=800.0 PL=0
MOVL C00601 V=800.0 PL=0
MOVL C00602 V=800.0 PL=0
MOVL C00603 V=800.0 PL=0
MOVL C00604 V=800.0 PL=0
MOVL C00605 V=800.0 PL=0
MOVL C00606 V=800.0 PL=0
MOVL C00607 V=800.0 PL=0
MOVL C00608 V=800.0 PL=0
MOVL C00609 V=800.0 PL=0
MOVL C00610 V=800.0 PL=0
MOVL C00611 V=800.0 PL=0
MOVL C00612 V=800.0 PL=0
MOVL C00613 V=800.0 PL=0
MOVL C00614 V=800.0 PL=0
MOVL C00615 V=800.0 PL=0
MOVL C00616 V=800.0 PL=0
MOVL C00617 V=800.0 PL=0
MOVL C00618 V=800.0 PL=0
MOVL C00619 V=800.0 PL=0
MOVL C00620 V=800.0 PL=0
MOVL C00621 V=800.0 PL=0
MOVL C00622 V=800.0 PL=0
MOVL C00623 V=800.0 PL=0
MOVL C00624 V=800.0 PL=0
MOVL C00625 V=800.0 PL=0
MOVL C00626 V=800.0 PL=0
MOVL C00627 V=800.0 PL=0
MOVL C00628 V=800.0 PL=0
MOVL C00629 V=800.0 PL=0
MOVL C00630 V=800.0 PL=0
MOVL C00631 V=800.0 PL=0
MOVL C00632 V=800.0 PL=0
MOVL C00633 V=800.0 PL=0
MOVL C00634 V=800.0 PL=0
MOVL C00635 V=800.0 PL=0
MOVL C00636 V=800.0 PL=0
MOVL C00637 V=800.0 PL=0
MOVL C00638 V=800.0 PL=0
MOVL C00639 V=800.0 PL=0
MOVL C00640 V=800.0 PL=0
MOVL C00641 V=800.0 PL=0
MOVL C00642 V=800.0 PL=0
MOVL C00643 V=800.0 PL=0
MOVL C00644 V=800.0 PL=0
MOVL C00645 V=800.0 PL=0
MOVL C00646 V=800.0 PL=0
MOVL C00647 V=800.0 PL=0
MOVL C00648 V=800.0 PL=0
MOVL C00649 V=800.0 PL=0
MOVL C00650 V=800.0 PL=0
MOVL C00651 V=800.0 PL=0
MOVL C00652 V=800.0 PL=0
MOVL C00653 V=800.0 PL=0
MOVL C00654 V=800.0 PL=0
MOVL C00655 V=800.0 PL=0
MOVL C00656 V=800.0 PL=0
MOVL C00657 V=800.0 PL=0
MOVL C00658 V=800.0 PL=0
MOVL C00659 V=800.0 PL=0
MOVL C00660 V=800.0 PL=0
MOVL C00661 V=800.0 PL=0
MOVL C00662 V=800.0 PL=0
MOVL C00663 V=800.0 PL=0
MOVL C00664 V=800.0 PL=0
MOVL C00665 V=800.0 PL=0
MOVL C00666 V=800.0 PL=0
MOVL C00667 V=800.0 PL=0
MOVL C00668 V=800.0 PL=0
MOVL C00669 V=800.0 PL=0
MOVL C00670 V=800.0 PL=0
MOVL C00671 V=800.0 PL=0
MOVL C00672 V=800.0 PL=0
MOVL C00673 V=800.0 PL=0
MOVL C00674 V=800.0 PL=0
MOVL C00675 V=800.0 PL=0
MOVL C00676 V=800.0 PL=0
MOVL C00677 V=800.0 PL=0
MOVL C00678 V=800.0 PL=0
MOVL C00679 V=800.0 PL=0
MOVL C00680 V=800.0 PL=0
MOVL C00681 V=800.0 PL=0
MOVL C00682 V=800.0 PL=0
MOVL C00683 V=800.0 PL=0
MOVL C00684 V=800.0 PL=0
MOVL C00685 V=800.0 PL=0
MOVL C00686 V=800.0 PL=0
MOVL C00687 V=800.0 PL=0
MOVL C00688 V=800.0 PL=0
MOVL C00689 V=800.0 PL=0
MOVL C00690 V=800.0 PL=0
MOVL C00691 V=800.0 PL=0
MOVL C00692 V=800.0 PL=0
MOVL C00693 V=800.0 PL=0
MOVL C00694 V=800.0 PL=0
MOVL C00695 V=800.0 PL=0
MOVL C00696 V=800.0 PL=0
MOVL C00697 V=800.0 PL=0
MOVL C00698 V=800.0 PL=0
MOVL C00699 V=800.0 PL=0
MOVL C00700 V=800.0 PL=0
MOVL C00701 V=800.0 PL=0
MOVL C00702 V=800.0 PL=0
MOVL C00703 V=800.0 PL=0
MOVL C00704 V=800.0 PL=0
MOVL C00705 V=800.0 PL=0
MOVL C00706 V=800.0 PL=0
MOVL C00707 V=800.0 PL=0
MOVL C00708 V=800.0 PL=0
MOVL C00709 V=800.0 PL=0
MOVL C00710 V=800.0 PL=0
MOVL C00711 V=800.0 PL=0
MOVL C00712 V=800.0 PL=0
MOVL C00713 V=800.0 PL=0
MOVL C00714 V=800.0 PL=0
MOVL C00715 V=800.0 PL=0
MOVL C00716 V=800.0 PL=0
MOVL C00717 V=800.0 PL=0
MOVL C00718 V=800.0 PL=0
MOVL C00719 V=800.0 PL=0
MOVL C00720 V=800.0 PL=0
MOVL C00721 V=800.0 PL=0
MOVL C00722 V=800.0 PL=0
MOVL C00723 V=800.0 PL=0
MOVL C00724 V=800.0 PL=0
MOVL C00725 V=800.0 PL=0
MOVL C00726 V=800.0 PL=0
MOVL C00727 V=800.0 PL=0
MOVL C00728 V=800.0 PL=0
MOVL C00729 V=800.0 PL=0
MOVL C00730 V=800.0 PL=0
MOVL C00731 V=800.0 PL=0
MOVL C00732 V=800.0 PL=0
MOVL C00733 V=800.0 PL=0
MOVL C00734 V=800.0 PL=0
MOVL C00735 V=800.0 PL=0
MOVL C00736 V=800.0 PL=0
MOVL C00737 V=800.0 PL=0
MOVL C00738 V=800.0 PL=0
MOVL C00739 V=800.0 PL=0
MOVL C00740 V=800.0 PL=0
MOVL C00741 V=800.0 PL=0
MOVL C00742 V=800.0 PL=0
MOVL C00743 V=800.0 PL=0
MOVL C00744 V=800.0 PL=0
MOVL C00745 V=800.0 PL=0
MOVL C00746 V=800.0 PL=0
MOVL C00747 V=800.0 PL=0
MOVL C00748 V=800.0 PL=0
MOVL C00749 V=800.0 PL=0
MOVL C00750 V=800.0 PL=0
MOVL C00751 V=800.0 PL=0
MOVL C00752 V=800.0 PL=0
MOVL C00753 V=800.0 PL=0
MOVL C00754 V=800.0 PL=0
MOVL C00755 V=800.0 PL=0
MOVL C00756 V=800.0 PL=0
MOVL C00757 V=800.0 PL=0
MOVL C00758 V=800.0 PL=0
MOVL C00759 V=800.0 PL=0
MOVL C00760 V=800.0 PL=0
MOVL C00761 V=800.0 PL=0
MOVL C00762 V=800.0 PL=0
MOVL C00763 V=800.0 PL=0
MOVL C00764 V=800.0 PL=0
MOVL C00765 V=800.0 PL=0
MOVL C00766 V=800.0 PL=0
MOVL C00767 V=800.0 PL=0
MOVL C00768 V=800.0 PL=0
MOVL C00769 V=800.0 PL=0
MOVL C00770 V=800.0 PL=0
MOVL C00771 V=800.0 PL=0
MOVL C00772 V=800.0 PL=0
MOVL C00773 V=800.0 PL=0
MOVL C00774 V=800.0 PL=0
MOVL C00775 V=800.0 PL=0
MOVL C00776 V=800.0 PL=0
MOVL C00777 V=800.0 PL=0
MOVL C00778 V=800.0 PL=0
MOVL C00779 V=800.0 PL=0
MOVL C00780 V=800.0 PL=0
MOVL C00781 V=800.0 PL=0
MOVL C00782 V=800.0 PL=0
MOVL C00783 V=800.0 PL=0
MOVL C00784 V=800.0 PL=0
MOVL C00785 V=800.0 PL=0
MOVL C00786 V=800.0 PL=0
MOVL C00787 V=800.0 PL=0
MOVL C00788 V=800.0 PL=0
MOVL C00789 V=800.0 PL=0
MOVL C00790 V=800.0 PL=0
MOVL C00791 V=800.0 PL=0
MOVL C00792 V=800.0 PL=0
MOVL C00793 V=800.0 PL=0
MOVL C00794 V=800.0 PL=0
MOVL C00795 V=800.0 PL=0
MOVL C00796 V=800.0 PL=0
MOVL C00797 V=800.0 PL=0
MOVL C00798 V=800.0 PL=0
MOVL C00799 V=800.0 PL=0
MOVL C00800 V=800.0 PL=0
MOVL C00801 V=800.0 PL=0
MOVL C00802 V=800.0 PL=0
MOVL C00803 V=800.0 PL=0
MOVL C00804 V=800.0 PL=0
MOVL C00805 V=800.0 PL=0
MOVL C00806 V=800.0 PL=0
MOVL C00807 V=800.0 PL=0
MOVL C00808 V=800.0 PL=0
MOVL C00809 V=800.0 PL=0
MOVL C00810 V=800.0 PL=0
MOVL C00811 V=800.0 PL=0
MOVL C00812 V=800.0 PL=0
MOVL C00813 V=800.0 PL=0
MOVL C00814 V=800.0 PL=0
MOVL C00815 V=800.0 PL=0
MOVL C00816 V=800.0 PL=0
MOVL C00817 V=800.0 PL=0
MOVL C00818 V=800.0 PL=0
MOVL C00819 V=800.0 PL=0
MOVL C00820 V=800.0 PL=0
MOVL C00821 V=800.0 PL=0
MOVL C00822 V=800.0 PL=0
MOVL C00823 V=800.0 PL=0
MOVL C00824 V=800.0 PL=0
MOVL C00825 V=800.0 PL=0
MOVL C00826 V=800.0 PL=0
MOVL C00827 V=800.0 PL=0
MOVL C00828 V=800.0 PL=0
MOVL C00829 V=800.0 PL=0
MOVL C00830 V=800.0 PL=0
MOVL C00831 V=800.0 PL=0
MOVL C00832 V=800.0 PL=0
MOVL C00833 V=800.0 PL=0
MOVL C00834 V=800.0 PL=0
MOVL C00835 V=800.0 PL=0
MOVL C00836 V=800.0 PL=0
MOVL C00837 V=800.0 PL=0
MOVL C00838 V=800.0 PL=0
MOVL C00839 V=800.0 PL=0
MOVL C00840 V=800.0 PL=0
MOVL C00841 V=800.0 PL=0
MOVL C00842 V=800.0 PL=0
MOVL C00843 V=800.0 PL=0
MOVL C00844 V=800.0 PL=0
MOVL C00845 V=800.0 PL=0
MOVL C00846 V=800.0 PL=0
MOVL C00847 V=800.0 PL=0
MOVL C00848 V=800.0 PL=0
MOVL C00849 V=800.0 PL=0
MOVL C00850 V=800.0 PL=0
MOVL C00851 V=800.0 PL=0
MOVL C00852 V=800.0 PL=0
MOVL C00853 V=800.0 PL=0
MOVL C00854 V=800.0 PL=0
MOVL C00855 V=800.0 PL=0
MOVL C00856 V=800.0 PL=0
MOVL C00857 V=800.0 PL=0
MOVL C00858 V=800.0 PL=0
MOVL C00859 V=800.0 PL=0
MOVL C00860 V=800.0 PL=0
MOVL C00861 V=800.0 PL=0
MOVL C00862 V=800.0 PL=0
MOVL C00863 V=800.0 PL=0
MOVL C00864 V=800.0 PL=0
MOVL C00865 V=800.0 PL=0
MOVL C00866 V=800.0 PL=0
MOVL C00867 V=800.0 PL=0
MOVL C00868 V=800.0 PL=0
MOVL C00869 V=800.0 PL=0
MOVL C00870 V=800.0 PL=0
MOVL C00871 V=800.0 PL=0
MOVL C00872 V=800.0 PL=0
MOVL C00873 V=800.0 PL=0
MOVL C00874 V=800.0 PL=0
MOVL C00875 V=800.0 PL=0
MOVL C00876 V=800.0 PL=0
MOVL C00877 V=800.0 PL=0
MOVL C00878 V=800.0 PL=0
MOVL C00879 V=800.0 PL=0
MOVL C00880 V=800.0 PL=0
MOVL C00881 V=800.0 PL=0
MOVL C00882 V=800.0 PL=0
MOVL C00883 V=800.0 PL=0
MOVL C00884 V=800.0 PL=0
MOVL C00885 V=800.0 PL=0
MOVL C00886 V=800.0 PL=0
MOVL C00887 V=800.0 PL=0
MOVL C00888 V=800.0 PL=0
MOVL C00889 V=800.0 PL=0
MOVL C00890 V=800.0 PL=0
MOVL C00891 V=800.0 PL=0
MOVL C00892 V=800.0 PL=0
MOVL C00893 V=800.0 PL=0
MOVL C00894 V=800.0 PL=0
MOVL C00895 V=800.0 PL=0
MOVL C00896 V=800.0 PL=0
MOVL C00897 V=800.0 PL=0
MOVL C00898 V=800.0 PL=0
MOVL C00899 V=800.0 PL=0
MOVL C00900 V=800.0 PL=0
MOVL C00901 V=800.0 PL=0
MOVL C00902 V=800.0 PL=0
MOVL C00903 V=800.0 PL=0
MOVL C00904 V=800.0 PL=0
MOVL C00905 V=800.0 PL=0
MOVL C00906 V=800.0 PL=0
MOVL C00907 V=800.0 PL=0
MOVL C00908 V=800.0 PL=0
MOVL C00909 V=800.0 PL=0
MOVL C00910 V=800.0 PL=0
MOVL C00911 V=800.0 PL=0
MOVL C00912 V=800.0 PL=0
MOVL C00913 V=800.0 PL=0
MOVL C00914 V=800.0 PL=0
MOVL C00915 V=800.0 PL=0
MOVL C00916 V=800.0 PL=0
MOVL C00917 V=800.0 PL=0
MOVL C00918 V=800.0 PL=0
MOVL C00919 V=800.0 PL=0
MOVL C00920 V=800.0 PL=0
MOVL C00921 V=800.0 PL=0
MOVL C00922 V=800.0 PL=0
MOVL C00923 V=800.0 PL=0
MOVL C00924 V=800.0 PL=0
MOVL C00925 V=800.0 PL=0
MOVL C00926 V=800.0 PL=0
MOVL C00927 V=800.0 PL=0
MOVL C00928 V=800.0 PL=0
MOVL C00929 V=800.0 PL=0
MOVL C00930 V=800.0 PL=0
MOVL C00931 V=800.0 PL=0
MOVL C00932 V=800.0 PL=0
MOVL C00933 V=800.0 PL=0
MOVL C00934 V=800.0 PL=0
MOVL C00935 V=800.0 PL=0
MOVL C00936 V=800.0 PL=0
MOVL C00937 V=800.0 PL=0
MOVL C00938 V=800.0 PL=0
MOVL C00939 V=800.0 PL=0
MOVL C00940 V=800.0 PL=0
MOVL C00941 V=800.0 PL=0
MOVL C00942 V=800.0 PL=0
MOVL C00943 V=800.0 PL=0
MOVL C00944 V=800.0 PL=0
MOVL C00945 V=800.0 PL=0
MOVL C00946 V=800.0 PL=0
MOVL C00947 V=800.0 PL=0
MOVL C00948 V=800.0 PL=0
MOVL C00949 V=800.0 PL=0
MOVL C00950 V=800.0 PL=0
MOVL C00951 V=800.0 PL=0
MOVL C00952 V=800.0 PL=0
MOVL C00953 V=800.0 PL=0
MOVL C00954 V=800.0 PL=0
MOVL C00955 V=800.0 PL=0
MOVL C00956 V=800.0 PL=0
MOVL C00957 V=800.0 PL=0
MOVL C00958 V=800.0 PL=0
MOVL C00959 V=800.0 PL=0
MOVL C00960 V=800.0 PL=0
MOVL C00961 V=800.0 PL=0
MOVL C00962 V=800.0 PL=0
MOVL C00963 V=800.0 PL=0
MOVL C00964 V=800.0 PL=0
MOVL C00965 V=800.0 PL=0
MOVL C00966 V=800.0 PL=0
MOVL C00967 V=800.0 PL=0
MOVL C00968 V=800.0 PL=0
MOVL C00969 V=800.0 PL=0
MOVL C00970 V=800.0 PL=0
MOVL C00971 V=800.0 PL=0
MOVL C00972 V=800.0 PL=0
MOVL C00973 V=800.0 PL=0
MOVL C00974 V=800.0 PL=0
MOVL C00975 V=800.0 PL=0
MOVL C00976 V=800.0 PL=0
MOVL C00977 V=800.0 PL=0
MOVL C00978 V=800.0 PL=0
MOVL C00979 V=800.0 PL=0
MOVL C00980 V=800.0 PL=0
MOVL C00981 V=800.0 PL=0
MOVL C00982 V=800.0 PL=0
MOVL C00983 V=800.0 PL=0
MOVL C00984 V=800.0 PL=0
MOVL C00985 V=800.0 PL=0
MOVL C00986 V=800.0 PL=0
MOVL C00987 V=800.0 PL=0
MOVL C00988 V=800.0 PL=0
MOVL C00989 V=800.0 PL=0
MOVL C00990 V=800.0 PL=0
MOVL C00991 V=800.0 PL=0
MOVL C00992 V=800.0 PL=0
MOVL C00993 V=800.0 PL=0
MOVL C00994 V=800.0 PL=0
MOVL C00995 V=800.0 PL=0
MOVL C00996 V=800.0 PL=0
MOVL C00997 V=800.0 PL=0
MOVL C00998 V=800.0 PL=0
MOVL C00999 V=800.0 PL=0
MOVL C01000 V=800.0 PL=0
MOVL C01001 V=800.0 PL=0
MOVL C01002 V=800.0 PL=0
MOVL C01003 V=800.0 PL=0
MOVL C01004 V=800.0 PL=0
MOVL C01005 V=800.0 PL=0
MOVL C01006 V=800.0 PL=0
MOVL C01007 V=800.0 PL=0
MOVL C01008 V=800.0 PL=0
MOVL C01009 V=800.0 PL=0
MOVL C01010 V=800.0 PL=0
MOVL C01011 V=800.0 PL=0
MOVL C01012 V=800.0 PL=0
MOVL C01013 V=800.0 PL=0
MOVL C01014 V=800.0 PL=0
MOVL C01015 V=800.0 PL=0
MOVL C01016 V=800.0 PL=0
MOVL C01017 V=800.0 PL=0
MOVL C01018 V=800.0 PL=0
MOVL C01019 V=800.0 PL=0
MOVL C01020 V=800.0 PL=0
MOVL C01021 V=800.0 PL=0
MOVL C01022 V=800.0 PL=0
MOVL C01023 V=800.0 PL=0
MOVL C01024 V=800.0 PL=0
MOVL C01025 V=800.0 PL=0
MOVL C01026 V=800.0 PL=0
MOVL C01027 V=800.0 PL=0
MOVL C01028 V=800.0 PL=0
MOVL C01029 V=800.0 PL=0
MOVL C01030 V=800.0 PL=0
MOVL C01031 V=800.0 PL=0
MOVL C01032 V=800.0 PL=0
MOVL C01033 V=800.0 PL=0
MOVL C01034 V=800.0 PL=0
MOVL C01035 V=800.0 PL=0
MOVL C01036 V=800.0 PL=0
MOVL C01037 V=800.0 PL=0
MOVL C01038 V=800.0 PL=0
MOVL C01039 V=800.0 PL=0
MOVL C01040 V=800.0 PL=0
MOVL C01041 V=800.0 PL=0
MOVL C01042 V=800.0 PL=0
MOVL C01043 V=800.0 PL=0
MOVL C01044 V=800.0 PL=0
MOVL C01045 V=800.0 PL=0
MOVL C01046 V=800.0 PL=0
MOVL C01047 V=800.0 PL=0
MOVL C01048 V=800.0 PL=0
MOVL C01049 V=800.0 PL=0
MOVL C01050 V=800.0 PL=0
MOVL C01051 V=800.0 PL=0
MOVL C01052 V=800.0 PL=0
MOVL C01053 V=800.0 PL=0
MOVL C01054 V=800.0 PL=0
MOVL C01055 V=800.0 PL=0
MOVL C01056 V=800.0 PL=0
MOVL C01057 V=800.0 PL=0
MOVL C01058 V=800.0 PL=0
MOVL C01059 V=800.0 PL=0
MOVL C01060 V=800.0 PL=0
MOVL C01061 V=800.0 PL=0
MOVL C01062 V=800.0 PL=0
MOVL C01063 V=800.0 PL=0
MOVL C01064 V=800.0 PL=0
MOVL C01065 V=800.0 PL=0
MOVL C01066 V=800.0 PL=0
MOVL C01067 V=800.0 PL=0
MOVL C01068 V=800.0 PL=0
MOVL C01069 V=800.0 PL=0
MOVL C01070 V=800.0 PL=0
MOVL C01071 V=800.0 PL=0
MOVL C01072 V=800.0 PL=0
MOVL C01073 V=800.0 PL=0
MOVL C01074 V=800.0 PL=0
MOVL C01075 V=800.0 PL=0
MOVL C01076 V=800.0 PL=0
MOVL C01077 V=800.0 PL=0
MOVL C01078 V=800.0 PL=0
MOVL C01079 V=800.0 PL=0
MOVL C01080 V=800.0 PL=0
MOVL C01081 V=800.0 PL=0
MOVL C01082 V=800.0 PL=0
MOVL C01083 V=800.0 PL=0
MOVL C01084 V=800.0 PL=0
MOVL C01085 V=800.0 PL=0
MOVL C01086 V=800.0 PL=0
MOVL C01087 V=800.0 PL=0
MOVL C01088 V=800.0 PL=0
MOVL C01089 V=800.0 PL=0
MOVL C01090 V=800.0 PL=0
MOVL C01091 V=800.0 PL=0
MOVL C01092 V=800.0 PL=0
MOVL C01093 V=800.0 PL=0
MOVL C01094 V=800.0 PL=0
MOVL C01095 V=800.0 PL=0
MOVL C01096 V=800.0 PL=0
MOVL C01097 V=800.0 PL=0
MOVL C01098 V=800.0 PL=0
MOVL C01099 V=800.0 PL=0
MOVL C01100 V=800.0 PL=0
MOVL C01101 V=800.0 PL=0
MOVL C01102 V=800.0 PL=0
MOVL C01103 V=800.0 PL=0
MOVL C01104 V=800.0 PL=0
MOVL C01105 V=800.0 PL=0
MOVL C01106 V=800.0 PL=0
MOVL C01107 V=800.0 PL=0
MOVL C01108 V=800.0 PL=0
MOVL C01109 V=800.0 PL=0
MOVL C01110 V=800.0 PL=0
MOVL C01111 V=800.0 PL=0
MOVL C01112 V=800.0 PL=0
MOVL C01113 V=800.0 PL=0
MOVL C01114 V=800.0 PL=0
MOVL C01115 V=800.0 PL=0
MOVL C01116 V=800.0 PL=0
MOVL C01117 V=800.0 PL=0
MOVL C01118 V=800.0 PL=0
MOVL C01119 V=800.0 PL=0
MOVL C01120 V=800.0 PL=0
MOVL C01121 V=800.0 PL=0
MOVL C01122 V=800.0 PL=0
MOVL C01123 V=800.0 PL=0
MOVL C01124 V=800.0 PL=0
MOVL C01125 V=800.0 PL=0
MOVL C01126 V=800.0 PL=0
MOVL C01127 V=800.0 PL=0
MOVL C01128 V=800.0 PL=0
MOVL C01129 V=800.0 PL=0
MOVL C01130 V=800.0 PL=0
MOVL C01131 V=800.0 PL=0
MOVL C01132 V=800.0 PL=0
MOVL C01133 V=800.0 PL=0
MOVL C01134 V=800.0 PL=0
MOVL C01135 V=800.0 PL=0
MOVL C01136 V=800.0 PL=0
MOVL C01137 V=800.0 PL=0
MOVL C01138 V=800.0 PL=0
MOVL C01139 V=800.0 PL=0
MOVL C01140 V=800.0 PL=0
MOVL C01141 V=800.0 PL=0
MOVL C01142 V=800.0 PL=0
MOVL C01143 V=800.0 PL=0
MOVL C01144 V=800.0 PL=0
MOVL C01145 V=800.0 PL=0
MOVL C01146 V=800.0 PL=0
MOVL C01147 V=800.0 PL=0
MOVL C01148 V=800.0 PL=0
MOVL C01149 V=800.0 PL=0
MOVL C01150 V=800.0 PL=0
MOVL C01151 V=800.0 PL=0
MOVL C01152 V=800.0 PL=0
MOVL C01153 V=800.0 PL=0
MOVL C01154 V=800.0 PL=0
MOVL C01155 V=800.0 PL=0
MOVL C01156 V=800.0 PL=0
MOVL C01157 V=800.0 PL=0
MOVL C01158 V=800.0 PL=0
MOVL C01159 V=800.0 PL=0
MOVL C01160 V=800.0 PL=0
MOVL C01161 V=800.0 PL=0
MOVL C01162 V=800.0 PL=0
MOVL C01163 V=800.0 PL=0
MOVL C01164 V=800.0 PL=0
MOVL C01165 V=800.0 PL=0
MOVL C01166 V=800.0 PL=0
MOVL C01167 V=800.0 PL=0
MOVL C01168 V=800.0 PL=0
MOVL C01169 V=800.0 PL=0
MOVL C01170 V=800.0 PL=0
MOVL C01171 V=800.0 PL=0
MOVL C01172 V=800.0 PL=0
MOVL C01173 V=800.0 PL=0
MOVL C01174 V=800.0 PL=0
MOVL C01175 V=800.0 PL=0
MOVL C01176 V=800.0 PL=0
MOVL C01177 V=800.0 PL=0
MOVL C01178 V=800.0 PL=0
MOVL C01179 V=800.0 PL=0
MOVL C01180 V=800.0 PL=0
MOVL C01181 V=800.0 PL=0
MOVL C01182 V=800.0 PL=0
MOVL C01183 V=800.0 PL=0
MOVL C01184 V=800.0 PL=0
MOVL C01185 V=800.0 PL=0
MOVL C01186 V=800.0 PL=0
MOVL C01187 V=800.0 PL=0
MOVL C01188 V=800.0 PL=0
MOVL C01189 V=800.0 PL=0
MOVL C01190 V=800.0 PL=0
MOVL C01191 V=800.0 PL=0
MOVL C01192 V=800.0 PL=0
MOVL C01193 V=800.0 PL=0
MOVL C01194 V=800.0 PL=0
MOVL C01195 V=800.0 PL=0
MOVL C01196 V=800.0 PL=0
MOVL C01197 V=800.0 PL=0
MOVL C01198 V=800.0 PL=0
MOVL C01199 V=800.0 PL=0
MOVL C01200 V=800.0 PL=0
MOVL C01201 V=800.0 PL=0
MOVL C01202 V=800.0 PL=0
MOVL C01203 V=800.0 PL=0
MOVL C01204 V=800.0 PL=0
MOVL C01205 V=800.0 PL=0
MOVL C01206 V=800.0 PL=0
MOVL C01207 V=800.0 PL=0
MOVL C01208 V=800.0 PL=0
MOVL C01209 V=800.0 PL=0
MOVL C01210 V=800.0 PL=0
MOVL C01211 V=800.0 PL=0
MOVL C01212 V=800.0 PL=0
MOVL C01213 V=800.0 PL=0
MOVL C01214 V=800.0 PL=0
MOVL C01215 V=800.0 PL=0
MOVL C01216 V=800.0 PL=0
MOVL C01217 V=800.0 PL=0
MOVL C01218 V=800.0 PL=0
MOVL C01219 V=800.0 PL=0
MOVL C01220 V=800.0 PL=0
MOVL C01221 V=800.0 PL=0
MOVL C01222 V=800.0 PL=0
MOVL C01223 V=800.0 PL=0
MOVL C01224 V=800.0 PL=0
MOVL C01225 V=800.0 PL=0
MOVL C01226 V=800.0 PL=0
MOVL C01227 V=800.0 PL=0
MOVL C01228 V=800.0 PL=0
MOVL C01229 V=800.0 PL=0
MOVL C01230 V=800.0 PL=0
MOVL C01231 V=800.0 PL=0
MOVL C01232 V=800.0 PL=0
MOVL C01233 V=800.0 PL=0
MOVL C01234 V=800.0 PL=0
MOVL C01235 V=800.0 PL=0
MOVL C01236 V=800.0 PL=0
MOVL C01237 V=800.0 PL=0
MOVL C01238 V=800.0 PL=0
MOVL C01239 V=800.0 PL=0
MOVL C01240 V=800.0 PL=0
MOVL C01241 V=800.0 PL=0
MOVL C01242 V=800.0 PL=0
MOVL C01243 V=800.0 PL=0
MOVL C01244 V=800.0 PL=0
MOVL C01245 V=800.0 PL=0
MOVL C01246 V=800.0 PL=0
MOVL C01247 V=800.0 PL=0
MOVL C01248 V=800.0 PL=0
MOVL C01249 V=800.0 PL=0
MOVL C01250 V=800.0 PL=0
MOVL C01251 V=800.0 PL=0
MOVL C01252 V=800.0 PL=0
MOVL C01253 V=800.0 PL=0
MOVL C01254 V=800.0 PL=0
MOVL C01255 V=800.0 PL=0
MOVL C01256 V=800.0 PL=0
MOVL C01257 V=800.0 PL=0
MOVL C01258 V=800.0 PL=0
MOVL C01259 V=800.0 PL=0
MOVL C01260 V=800.0 PL=0
MOVL C01261 V=800.0 PL=0
MOVL C01262 V=800.0 PL=0
MOVL C01263 V=800.0 PL=0
MOVL C01264 V=800.0 PL=0
MOVL C01265 V=800.0 PL=0
MOVL C01266 V=800.0 PL=0
MOVL C01267 V=800.0 PL=0
MOVL C01268 V=800.0 PL=0
MOVL C01269 V=800.0 PL=0
MOVL C01270 V=800.0 PL=0
MOVL C01271 V=800.0 PL=0
MOVL C01272 V=800.0 PL=0
MOVL C01273 V=800.0 PL=0
MOVL C01274 V=800.0 PL=0
MOVL C01275 V=800.0 PL=0
MOVL C01276 V=800.0 PL=0
MOVL C01277 V=800.0 PL=0
MOVL C01278 V=800.0 PL=0
MOVL C01279 V=800.0 PL=0
MOVL C01280 V=800.0 PL=0
MOVL C01281 V=800.0 PL=0
MOVL C01282 V=800.0 PL=0
MOVL C01283 V=800.0 PL=0
MOVL C01284 V=800.0 PL=0
MOVL C01285 V=800.0 PL=0
MOVL C01286 V=800.0 PL=0
MOVL C01287 V=800.0 PL=0
MOVL C01288 V=800.0 PL=0
MOVL C01289 V=800.0 PL=0
MOVL C01290 V=800.0 PL=0
MOVL C01291 V=800.0 PL=0
MOVL C01292 V=800.0 PL=0
MOVL C01293 V=800.0 PL=0
MOVL C01294 V=800.0 PL=0
MOVL C01295 V=800.0 PL=0
MOVL C01296 V=800.0 PL=0
MOVL C01297 V=800.0 PL=0
MOVL C01298 V=800.0 PL=0
MOVL C01299 V=800.0 PL=0
MOVL C01300 V=800.0 PL=0
MOVL C01301 V=800.0 PL=0
MOVL C01302 V=800.0 PL=0
MOVL C01303 V=800.0 PL=0
MOVL C01304 V=800.0 PL=0
MOVL C01305 V=800.0 PL=0
MOVL C01306 V=800.0 PL=0
MOVL C01307 V=800.0 PL=0
MOVL C01308 V=800.0 PL=0
MOVL C01309 V=800.0 PL=0
MOVL C01310 V=800.0 PL=0
MOVL C01311 V=800.0 PL=0
MOVL C01312 V=800.0 PL=0
MOVL C01313 V=800.0 PL=0
MOVL C01314 V=800.0 PL=0
MOVL C01315 V=800.0 PL=0
MOVL C01316 V=800.0 PL=0
MOVL C01317 V=800.0 PL=0
MOVL C01318 V=800.0 PL=0
MOVL C01319 V=800.0 PL=0
MOVL C01320 V=800.0 PL=0
MOVL C01321 V=800.0 PL=0
MOVL C01322 V=800.0 PL=0
MOVL C01323 V=800.0 PL=0
MOVL C01324 V=800.0 PL=0
MOVL C01325 V=800.0 PL=0
MOVL C01326 V=800.0 PL=0
MOVL C01327 V=800.0 PL=0
MOVL C01328 V=800.0 PL=0
MOVL C01329 V=800.0 PL=0
MOVL C01330 V=800.0 PL=0
MOVL C01331 V=800.0 PL=0
MOVL C01332 V=800.0 PL=0
MOVL C01333 V=800.0 PL=0
MOVL C01334 V=800.0 PL=0
MOVL C01335 V=800.0 PL=0
MOVL C01336 V=800.0 PL=0
MOVL C01337 V=800.0 PL=0
MOVL C01338 V=800.0 PL=0
MOVL C01339 V=800.0 PL=0
MOVL C01340 V=800.0 PL=0
MOVL C01341 V=800.0 PL=0
MOVL C01342 V=800.0 PL=0
MOVL C01343 V=800.0 PL=0
MOVL C01344 V=800.0 PL=0
MOVL C01345 V=800.0 PL=0
MOVL C01346 V=800.0 PL=0
MOVL C01347 V=800.0 PL=0
MOVL C01348 V=800.0 PL=0
MOVL C01349 V=800.0 PL=0
MOVL C01350 V=800.0 PL=0
MOVL C01351 V=800.0 PL=0
MOVL C01352 V=800.0 PL=0
MOVL C01353 V=800.0 PL=0
MOVL C01354 V=800.0 PL=0
MOVL C01355 V=800.0 PL=0
MOVL C01356 V=800.0 PL=0
MOVL C01357 V=800.0 PL=0
MOVL C01358 V=800.0 PL=0
MOVL C01359 V=800.0 PL=0
MOVL C01360 V=800.0 PL=0
MOVL C01361 V=800.0 PL=0
MOVL C01362 V=800.0 PL=0
MOVL C01363 V=800.0 PL=0
MOVL C01364 V=800.0 PL=0
MOVL C01365 V=800.0 PL=0
MOVL C01366 V=800.0 PL=0
MOVL C01367 V=800.0 PL=0
MOVL C01368 V=800.0 PL=0
MOVL C01369 V=800.0 PL=0
MOVL C01370 V=800.0 PL=0
MOVL C01371 V=800.0 PL=0
MOVL C01372 V=800.0 PL=0
MOVL C01373 V=800.0 PL=0
MOVL C01374 V=800.0 PL=0
MOVL C01375 V=800.0 PL=0
MOVL C01376 V=800.0 PL=0
MOVL C01377 V=800.0 PL=0
MOVL C01378 V=800.0 PL=0
MOVL C01379 V=800.0 PL=0
MOVL C01380 V=800.0 PL=0
MOVL C01381 V=800.0 PL=0
MOVL C01382 V=800.0 PL=0
MOVL C01383 V=800.0 PL=0
MOVL C01384 V=800.0 PL=0
MOVL C01385 V=800.0 PL=0
MOVL C01386 V=800.0 PL=0
MOVL C01387 V=800.0 PL=0
MOVL C01388 V=800.0 PL=0
MOVL C01389 V=800.0 PL=0
MOVL C01390 V=800.0 PL=0
MOVL C01391 V=800.0 PL=0
MOVL C01392 V=800.0 PL=0
MOVL C01393 V=800.0 PL=0
MOVL C01394 V=800.0 PL=0
MOVL C01395 V=800.0 PL=0
MOVL C01396 V=800.0 PL=0
MOVL C01397 V=800.0 PL=0
MOVL C01398 V=800.0 PL=0
MOVL C01399 V=800.0 PL=0
MOVL C01400 V=800.0 PL=0
MOVL C01401 V=800.0 PL=0
MOVL C01402 V=800.0 PL=0
MOVL C01403 V=800.0 PL=0
MOVL C01404 V=800.0 PL=0
MOVL C01405 V=800.0 PL=0
MOVL C01406 V=800.0 PL=0
MOVL C01407 V=800.0 PL=0
MOVL C01408 V=800.0 PL=0
MOVL C01409 V=800.0 PL=0
MOVL C01410 V=800.0 PL=0
MOVL C01411 V=800.0 PL=0
MOVL C01412 V=800.0 PL=0
MOVL C01413 V=800.0 PL=0
MOVL C01414 V=800.0 PL=0
MOVL C01415 V=800.0 PL=0
MOVL C01416 V=800.0 PL=0
MOVL C01417 V=800.0 PL=0
MOVL C01418 V=800.0 PL=0
MOVL C01419 V=800.0 PL=0
MOVL C01420 V=800.0 PL=0
MOVL C01421 V=800.0 PL=0
MOVL C01422 V=800.0 PL=0
MOVL C01423 V=800.0 PL=0
MOVL C01424 V=800.0 PL=0
MOVL C01425 V=800.0 PL=0
MOVL C01426 V=800.0 PL=0
MOVL C01427 V=800.0 PL=0
MOVL C01428 V=800.0 PL=0
MOVL C01429 V=800.0 PL=0
MOVL C01430 V=800.0 PL=0
MOVL C01431 V=800.0 PL=0
MOVL C01432 V=800.0 PL=0
MOVL C01433 V=800.0 PL=0
MOVL C01434 V=800.0 PL=0
MOVL C01435 V=800.0 PL=0
MOVL C01436 V=800.0 PL=0
MOVL C01437 V=800.0 PL=0
MOVL C01438 V=800.0 PL=0
MOVL C01439 V=800.0 PL=0
MOVL C01440 V=800.0 PL=0
MOVL C01441 V=800.0 PL=0
MOVL C01442 V=800.0 PL=0
MOVL C01443 V=800.0 PL=0
MOVL C01444 V=800.0 PL=0
MOVL C01445 V=800.0 PL=0
MOVL C01446 V=800.0 PL=0
MOVL C01447 V=800.0 PL=0
MOVL C01448 V=800.0 PL=0
MOVL C01449 V=800.0 PL=0
MOVL C01450 V=800.0 PL=0
MOVL C01451 V=800.0 PL=0
MOVL C01452 V=800.0 PL=0
MOVL C01453 V=800.0 PL=0
MOVL C01454 V=800.0 PL=0
MOVL C01455 V=800.0 PL=0
MOVL C01456 V=800.0 PL=0
MOVL C01457 V=800.0 PL=0
MOVL C01458 V=800.0 PL=0
MOVL C01459 V=800.0 PL=0
MOVL C01460 V=800.0 PL=0
MOVL C01461 V=800.0 PL=0
MOVL C01462 V=800.0 PL=0
MOVL C01463 V=800.0 PL=0
MOVL C01464 V=800.0 PL=0
MOVL C01465 V=800.0 PL=0
MOVL C01466 V=800.0 PL=0
MOVL C01467 V=800.0 PL=0
MOVL C01468 V=800.0 PL=0
MOVL C01469 V=800.0 PL=0
MOVL C01470 V=800.0 PL=0
MOVL C01471 V=800.0 PL=0
MOVL C01472 V=800.0 PL=0
MOVL C01473 V=800.0 PL=0
MOVL C01474 V=800.0 PL=0
MOVL C01475 V=800.0 PL=0
MOVL C01476 V=800.0 PL=0
MOVL C01477 V=800.0 PL=0
MOVL C01478 V=800.0 PL=0
MOVL C01479 V=800.0 PL=0
MOVL C01480 V=800.0 PL=0
MOVL C01481 V=800.0 PL=0
MOVL C01482 V=800.0 PL=0
MOVL C01483 V=800.0 PL=0
MOVL C01484 V=800.0 PL=0
MOVL C01485 V=800.0 PL=0
MOVL C01486 V=800.0 PL=0
MOVL C01487 V=800.0 PL=0
MOVL C01488 V=800.0 PL=0
MOVL C01489 V=800.0 PL=0
MOVL C01490 V=800.0 PL=0
MOVL C01491 V=800.0 PL=0
MOVL C01492 V=800.0 PL=0
MOVL C01493 V=800.0 PL=0
MOVL C01494 V=800.0 PL=0
MOVL C01495 V=800.0 PL=0
MOVL C01496 V=800.0 PL=0
MOVL C01497 V=800.0 PL=0
MOVL C01498 V=800.0 PL=0
MOVL C01499 V=800.0 PL=0
MOVL C01500 V=800.0 PL=0
MOVL C01501 V=800.0 PL=0
MOVL C01502 V=800.0 PL=0
MOVL C01503 V=800.0 PL=0
MOVL C01504 V=800.0 PL=0
MOVL C01505 V=800.0 PL=0
MOVL C01506 V=800.0 PL=0
MOVL C01507 V=800.0 PL=0
MOVL C01508 V=800.0 PL=0
MOVL C01509 V=800.0 PL=0
MOVL C01510 V=800.0 PL=0
MOVL C01511 V=800.0 PL=0
MOVL C01512 V=800.0 PL=0
MOVL C01513 V=800.0 PL=0
MOVL C01514 V=800.0 PL=0
MOVL C01515 V=800.0 PL=0
MOVL C01516 V=800.0 PL=0
MOVL C01517 V=800.0 PL=0
MOVL C01518 V=800.0 PL=0
MOVL C01519 V=800.0 PL=0
MOVL C01520 V=800.0 PL=0
MOVL C01521 V=800.0 PL=0
MOVL C01522 V=800.0 PL=0
MOVL C01523 V=800.0 PL=0
MOVL C01524 V=800.0 PL=0
MOVL C01525 V=800.0 PL=0
MOVL C01526 V=800.0 PL=0
MOVL C01527 V=800.0 PL=0
MOVL C01528 V=800.0 PL=0
MOVL C01529 V=800.0 PL=0
MOVL C01530 V=800.0 PL=0
MOVL C01531 V=800.0 PL=0
MOVL C01532 V=800.0 PL=0
MOVL C01533 V=800.0 PL=0
MOVL C01534 V=800.0 PL=0
MOVL C01535 V=800.0 PL=0
MOVL C01536 V=800.0 PL=0
MOVL C01537 V=800.0 PL=0
MOVL C01538 V=800.0 PL=0
MOVL C01539 V=800.0 PL=0
MOVL C01540 V=800.0 PL=0
MOVL C01541 V=800.0 PL=0
MOVL C01542 V=800.0 PL=0
MOVL C01543 V=800.0 PL=0
MOVL C01544 V=800.0 PL=0
MOVL C01545 V=800.0 PL=0
MOVL C01546 V=800.0 PL=0
MOVL C01547 V=800.0 PL=0
MOVL C01548 V=800.0 PL=0
MOVL C01549 V=800.0 PL=0
MOVL C01550 V=800.0 PL=0
MOVL C01551 V=800.0 PL=0
MOVL C01552 V=800.0 PL=0
MOVL C01553 V=800.0 PL=0
MOVL C01554 V=800.0 PL=0
MOVL C01555 V=800.0 PL=0
MOVL C01556 V=800.0 PL=0
MOVL C01557 V=800.0 PL=0
MOVL C01558 V=800.0 PL=0
MOVL C01559 V=800.0 PL=0
MOVL C01560 V=800.0 PL=0
MOVL C01561 V=800.0 PL=0
MOVL C01562 V=800.0 PL=0
MOVL C01563 V=800.0 PL=0
MOVL C01564 V=800.0 PL=0
MOVL C01565 V=800.0 PL=0
MOVL C01566 V=800.0 PL=0
MOVL C01567 V=800.0 PL=0
MOVL C01568 V=800.0 PL=0
MOVL C01569 V=800.0 PL=0
MOVL C01570 V=800.0 PL=0
MOVL C01571 V=800.0 PL=0
MOVL C01572 V=800.0 PL=0
MOVL C01573 V=800.0 PL=0
MOVL C01574 V=800.0 PL=0
MOVL C01575 V=800.0 PL=0
MOVL C01576 V=800.0 PL=0
MOVL C01577 V=800.0 PL=0
MOVL C01578 V=800.0 PL=0
MOVL C01579 V=800.0 PL=0
MOVL C01580 V=800.0 PL=0
MOVL C01581 V=800.0 PL=0
MOVL C01582 V=800.0 PL=0
MOVL C01583 V=800.0 PL=0
MOVL C01584 V=800.0 PL=0
MOVL C01585 V=800.0 PL=0
MOVL C01586 V=800.0 PL=0
MOVL C01587 V=800.0 PL=0
MOVL C01588 V=800.0 PL=0
MOVL C01589 V=800.0 PL=0
MOVL C01590 V=800.0 PL=0
MOVL C01591 V=800.0 PL=0
MOVL C01592 V=800.0 PL=0
MOVL C01593 V=800.0 PL=0
MOVL C01594 V=800.0 PL=0
MOVL C01595 V=800.0 PL=0
MOVL C01596 V=800.0 PL=0
MOVL C01597 V=800.0 PL=0
MOVL C01598 V=800.0 PL=0
MOVL C01599 V=800.0 PL=0
MOVL C01600 V=800.0 PL=0
MOVL C01601 V=800.0 PL=0
MOVL C01602 V=800.0 PL=0
MOVL C01603 V=800.0 PL=0
MOVL C01604 V=800.0 PL=0
MOVL C01605 V=800.0 PL=0
MOVL C01606 V=800.0 PL=0
MOVL C01607 V=800.0 PL=0
MOVL C01608 V=800.0 PL=0
MOVL C01609 V=800.0 PL=0
MOVL C01610 V=800.0 PL=0
MOVL C01611 V=800.0 PL=0
MOVL C01612 V=800.0 PL=0
MOVL C01613 V=800.0 PL=0
MOVL C01614 V=800.0 PL=0
MOVL C01615 V=800.0 PL=0
MOVL C01616 V=800.0 PL=0
MOVL C01617 V=800.0 PL=0
MOVL C01618 V=800.0 PL=0
MOVL C01619 V=800.0 PL=0
MOVL C01620 V=800.0 PL=0
MOVL C01621 V=800.0 PL=0
MOVL C01622 V=800.0 PL=0
MOVL C01623 V=800.0 PL=0
MOVL C01624 V=800.0 PL=0
MOVL C01625 V=800.0 PL=0
MOVL C01626 V=800.0 PL=0
MOVL C01627 V=800.0 PL=0
MOVL C01628 V=800.0 PL=0
MOVL C01629 V=800.0 PL=0
MOVL C01630 V=800.0 PL=0
MOVL C01631 V=800.0 PL=0
MOVL C01632 V=800.0 PL=0
MOVL C01633 V=800.0 PL=0
MOVL C01634 V=800.0 PL=0
MOVL C01635 V=800.0 PL=0
MOVL C01636 V=800.0 PL=0
MOVL C01637 V=800.0 PL=0
MOVL C01638 V=800.0 PL=0
MOVL C01639 V=800.0 PL=0
MOVL C01640 V=800.0 PL=0
MOVL C01641 V=800.0 PL=0
MOVL C01642 V=800.0 PL=0
MOVL C01643 V=800.0 PL=0
MOVL C01644 V=800.0 PL=0
MOVL C01645 V=800.0 PL=0
MOVL C01646 V=800.0 PL=0
MOVL C01647 V=800.0 PL=0
MOVL C01648 V=800.0 PL=0
MOVL C01649 V=800.0 PL=0
MOVL C01650 V=800.0 PL=0
MOVL C01651 V=800.0 PL=0
MOVL C01652 V=800.0 PL=0
MOVL C01653 V=800.0 PL=0
MOVL C01654 V=800.0 PL=0
MOVL C01655 V=800.0 PL=0
MOVL C01656 V=800.0 PL=0
MOVL C01657 V=800.0 PL=0
MOVL C01658 V=800.0 PL=0
MOVL C01659 V=800.0 PL=0
MOVL C01660 V=800.0 PL=0
MOVL C01661 V=800.0 PL=0
MOVL C01662 V=800.0 PL=0
MOVL C01663 V=800.0 PL=0
MOVL C01664 V=800.0 PL=0
MOVL C01665 V=800.0 PL=0
MOVL C01666 V=800.0 PL=0
MOVL C01667 V=800.0 PL=0
MOVL C01668 V=800.0 PL=0
MOVL C01669 V=800.0 PL=0
MOVL C01670 V=800.0 PL=0
MOVL C01671 V=800.0 PL=0
MOVL C01672 V=800.0 PL=0
MOVL C01673 V=800.0 PL=0
MOVL C01674 V=800.0 PL=0
MOVL C01675 V=800.0 PL=0
MOVL C01676 V=800.0 PL=0
MOVL C01677 V=800.0 PL=0
MOVL C01678 V=800.0 PL=0
MOVL C01679 V=800.0 PL=0
MOVL C01680 V=800.0 PL=0
MOVL C01681 V=800.0 PL=0
MOVL C01682 V=800.0 PL=0
MOVL C01683 V=800.0 PL=0
MOVL C01684 V=800.0 PL=0
MOVL C01685 V=800.0 PL=0
MOVL C01686 V=800.0 PL=0
MOVL C01687 V=800.0 PL=0
MOVL C01688 V=800.0 PL=0
MOVL C01689 V=800.0 PL=0
MOVL C01690 V=800.0 PL=0
MOVL C01691 V=800.0 PL=0
MOVL C01692 V=800.0 PL=0
MOVL C01693 V=800.0 PL=0
MOVL C01694 V=800.0 PL=0
MOVL C01695 V=800.0 PL=0
MOVL C01696 V=800.0 PL=0
MOVL C01697 V=800.0 PL=0
MOVL C01698 V=800.0 PL=0
MOVL C01699 V=800.0 PL=0
MOVL C01700 V=800.0 PL=0
MOVL C01701 V=800.0 PL=0
MOVL C01702 V=800.0 PL=0
MOVL C01703 V=800.0 PL=0
MOVL C01704 V=800.0 PL=0
MOVL C01705 V=800.0 PL=0
MOVL C01706 V=800.0 PL=0
MOVL C01707 V=800.0 PL=0
MOVL C01708 V=800.0 PL=0
MOVL C01709 V=800.0 PL=0
MOVL C01710 V=800.0 PL=0
MOVL C01711 V=800.0 PL=0
MOVL C01712 V=800.0 PL=0
MOVL C01713 V=800.0 PL=0
MOVL C01714 V=800.0 PL=0
MOVL C01715 V=800.0 PL=0
MOVL C01716 V=800.0 PL=0
MOVL C01717 V=800.0 PL=0
MOVL C01718 V=800.0 PL=0
MOVL C01719 V=800.0 PL=0
MOVL C01720 V=800.0 PL=0
MOVL C01721 V=800.0 PL=0
MOVL C01722 V=800.0 PL=0
MOVL C01723 V=800.0 PL=0
MOVL C01724 V=800.0 PL=0
MOVL C01725 V=800.0 PL=0
MOVL C01726 V=800.0 PL=0
MOVL C01727 V=800.0 PL=0
MOVL C01728 V=800.0 PL=0
MOVL C01729 V=800.0 PL=0
MOVL C01730 V=800.0 PL=0
MOVL C01731 V=800.0 PL=0
MOVL C01732 V=800.0 PL=0
MOVL C01733 V=800.0 PL=0
MOVL C01734 V=800.0 PL=0
MOVL C01735 V=800.0 PL=0
MOVL C01736 V=800.0 PL=0
MOVL C01737 V=800.0 PL=0
MOVL C01738 V=800.0 PL=0
MOVL C01739 V=800.0 PL=0
MOVL C01740 V=800.0 PL=0
MOVL C01741 V=800.0 PL=0
MOVL C01742 V=800.0 PL=0
MOVL C01743 V=800.0 PL=0
MOVL C01744 V=800.0 PL=0
MOVL C01745 V=800.0 PL=0
MOVL C01746 V=800.0 PL=0
MOVL C01747 V=800.0 PL=0
MOVL C01748 V=800.0 PL=0
MOVL C01749 V=800.0 PL=0
MOVL C01750 V=800.0 PL=0
MOVL C01751 V=800.0 PL=0
MOVL C01752 V=800.0 PL=0
MOVL C01753 V=800.0 PL=0
MOVL C01754 V=800.0 PL=0
MOVL C01755 V=800.0 PL=0
MOVL C01756 V=800.0 PL=0
MOVL C01757 V=800.0 PL=0
MOVL C01758 V=800.0 PL=0
MOVL C01759 V=800.0 PL=0
MOVL C01760 V=800.0 PL=0
MOVL C01761 V=800.0 PL=0
MOVL C01762 V=800.0 PL=0
MOVL C01763 V=800.0 PL=0
MOVL C01764 V=800.0 PL=0
MOVL C01765 V=800.0 PL=0
MOVL C01766 V=800.0 PL=0
MOVL C01767 V=800.0 PL=0
MOVL C01768 V=800.0 PL=0
MOVL C01769 V=800.0 PL=0
MOVL C01770 V=800.0 PL=0
MOVL C01771 V=800.0 PL=0
MOVL C01772 V=800.0 PL=0
MOVL C01773 V=800.0 PL=0
MOVL C01774 V=800.0 PL=0
MOVL C01775 V=800.0 PL=0
MOVL C01776 V=800.0 PL=0
MOVL C01777 V=800.0 PL=0
MOVL C01778 V=800.0 PL=0
MOVL C01779 V=800.0 PL=0
MOVL C01780 V=800.0 PL=0
MOVL C01781 V=800.0 PL=0
MOVL C01782 V=800.0 PL=0
MOVL C01783 V=800.0 PL=0
MOVL C01784 V=800.0 PL=0
MOVL C01785 V=800.0 PL=0
MOVL C01786 V=800.0 PL=0
MOVL C01787 V=800.0 PL=0
MOVL C01788 V=800.0 PL=0
MOVL C01789 V=800.0 PL=0
MOVL C01790 V=800.0 PL=0
MOVL C01791 V=800.0 PL=0
MOVL C01792 V=800.0 PL=0
MOVL C01793 V=800.0 PL=0
MOVL C01794 V=800.0 PL=0
MOVL C01795 V=800.0 PL=0
MOVL C01796 V=800.0 PL=0
MOVL C01797 V=800.0 PL=0
MOVL C01798 V=800.0 PL=0
MOVL C01799 V=800.0 PL=0
MOVL C01800 V=800.0 PL=0
MOVL C01801 V=800.0 PL=0
MOVL C01802 V=800.0 PL=0
MOVL C01803 V=800.0 PL=0
MOVL C01804 V=800.0 PL=0
MOVL C01805 V=800.0 PL=0
MOVL C01806 V=800.0 PL=0
MOVL C01807 V=800.0 PL=0
MOVL C01808 V=800.0 PL=0
MOVL C01809 V=800.0 PL=0
MOVL C01810 V=800.0 PL=0
MOVL C01811 V=800.0 PL=0
MOVL C01812 V=800.0 PL=0
MOVL C01813 V=800.0 PL=0
MOVL C01814 V=800.0 PL=0
MOVL C01815 V=800.0 PL=0
MOVL C01816 V=800.0 PL=0
MOVL C01817 V=800.0 PL=0
MOVL C01818 V=800.0 PL=0
MOVL C01819 V=800.0 PL=0
MOVL C01820 V=800.0 PL=0
MOVL C01821 V=800.0 PL=0
MOVL C01822 V=800.0 PL=0
MOVL C01823 V=800.0 PL=0
MOVL C01824 V=800.0 PL=0
MOVL C01825 V=800.0 PL=0
MOVL C01826 V=800.0 PL=0
MOVL C01827 V=800.0 PL=0
MOVL C01828 V=800.0 PL=0
MOVL C01829 V=800.0 PL=0
MOVL C01830 V=800.0 PL=0
MOVL C01831 V=800.0 PL=0
MOVL C01832 V=800.0 PL=0
MOVL C01833 V=800.0 PL=0
MOVL C01834 V=800.0 PL=0
MOVL C01835 V=800.0 PL=0
MOVL C01836 V=800.0 PL=0
MOVL C01837 V=800.0 PL=0
MOVL C01838 V=800.0 PL=0
MOVL C01839 V=800.0 PL=0
MOVL C01840 V=800.0 PL=0
MOVL C01841 V=800.0 PL=0
MOVL C01842 V=800.0 PL=0
MOVL C01843 V=800.0 PL=0
MOVL C01844 V=800.0 PL=0
MOVL C01845 V=800.0 PL=0
MOVL C01846 V=800.0 PL=0
MOVL C01847 V=800.0 PL=0
MOVL C01848 V=800.0 PL=0
MOVL C01849 V=800.0 PL=0
MOVL C01850 V=800.0 PL=0
MOVL C01851 V=800.0 PL=0
MOVL C01852 V=800.0 PL=0
MOVL C01853 V=800.0 PL=0
MOVL C01854 V=800.0 PL=0
MOVL C01855 V=800.0 PL=0
MOVL C01856 V=800.0 PL=0
MOVL C01857 V=800.0 PL=0
MOVL C01858 V=800.0 PL=0
MOVL C01859 V=800.0 PL=0
MOVL C01860 V=800.0 PL=0
MOVL C01861 V=800.0 PL=0
MOVL C01862 V=800.0 PL=0
MOVL C01863 V=800.0 PL=0
MOVL C01864 V=800.0 PL=0
MOVL C01865 V=800.0 PL=0
MOVL C01866 V=800.0 PL=0
MOVL C01867 V=800.0 PL=0
MOVL C01868 V=800.0 PL=0
MOVL C01869 V=800.0 PL=0
MOVL C01870 V=800.0 PL=0
MOVL C01871 V=800.0 PL=0
MOVL C01872 V=800.0 PL=0
MOVL C01873 V=800.0 PL=0
MOVL C01874 V=800.0 PL=0
MOVL C01875 V=800.0 PL=0
MOVL C01876 V=800.0 PL=0
MOVL C01877 V=800.0 PL=0
MOVL C01878 V=800.0 PL=0
MOVL C01879 V=800.0 PL=0
MOVL C01880 V=800.0 PL=0
MOVL C01881 V=800.0 PL=0
MOVL C01882 V=800.0 PL=0
MOVL C01883 V=800.0 PL=0
MOVL C01884 V=800.0 PL=0
MOVL C01885 V=800.0 PL=0
MOVL C01886 V=800.0 PL=0
MOVL C01887 V=800.0 PL=0
MOVL C01888 V=800.0 PL=0
MOVL C01889 V=800.0 PL=0
MOVL C01890 V=800.0 PL=0
MOVL C01891 V=800.0 PL=0
MOVL C01892 V=800.0 PL=0
MOVL C01893 V=800.0 PL=0
MOVL C01894 V=800.0 PL=0
MOVL C01895 V=800.0 PL=0
MOVL C01896 V=800.0 PL=0
MOVL C01897 V=800.0 PL=0
MOVL C01898 V=800.0 PL=0
MOVL C01899 V=800.0 PL=0
MOVL C01900 V=800.0 PL=0
MOVL C01901 V=800.0 PL=0
MOVL C01902 V=800.0 PL=0
MOVL C01903 V=800.0 PL=0
MOVL C01904 V=800.0 PL=0
MOVL C01905 V=800.0 PL=0
MOVL C01906 V=800.0 PL=0
MOVL C01907 V=800.0 PL=0
MOVL C01908 V=800.0 PL=0
MOVL C01909 V=800.0 PL=0
MOVL C01910 V=800.0 PL=0
MOVL C01911 V=800.0 PL=0
MOVL C01912 V=800.0 PL=0
MOVL C01913 V=800.0 PL=0
MOVL C01914 V=800.0 PL=0
MOVL C01915 V=800.0 PL=0
MOVL C01916 V=800.0 PL=0
MOVL C01917 V=800.0 PL=0
MOVL C01918 V=800.0 PL=0
MOVL C01919 V=800.0 PL=0
MOVL C01920 V=800.0 PL=0
MOVL C01921 V=800.0 PL=0
MOVL C01922 V=800.0 PL=0
MOVL C01923 V=800.0 PL=0
MOVL C01924 V=800.0 PL=0
MOVL C01925 V=800.0 PL=0
MOVL C01926 V=800.0 PL=0
MOVL C01927 V=800.0 PL=0
MOVL C01928 V=800.0 PL=0
MOVL C01929 V=800.0 PL=0
MOVL C01930 V=800.0 PL=0
MOVL C01931 V=800.0 PL=0
MOVL C01932 V=800.0 PL=0
MOVL C01933 V=800.0 PL=0
MOVL C01934 V=800.0 PL=0
MOVL C01935 V=800.0 PL=0
MOVL C01936 V=800.0 PL=0
MOVL C01937 V=800.0 PL=0
MOVL C01938 V=800.0 PL=0
MOVL C01939 V=800.0 PL=0
MOVL C01940 V=800.0 PL=0
MOVL C01941 V=800.0 PL=0
MOVL C01942 V=800.0 PL=0
MOVL C01943 V=800.0 PL=0
MOVL C01944 V=800.0 PL=0
MOVL C01945 V=800.0 PL=0
MOVL C01946 V=800.0 PL=0
MOVL C01947 V=800.0 PL=0
MOVL C01948 V=800.0 PL=0
MOVL C01949 V=800.0 PL=0
MOVL C01950 V=800.0 PL=0
MOVL C01951 V=800.0 PL=0
MOVL C01952 V=800.0 PL=0
MOVL C01953 V=800.0 PL=0
MOVL C01954 V=800.0 PL=0
MOVL C01955 V=800.0 PL=0
MOVL C01956 V=800.0 PL=0
MOVL C01957 V=800.0 PL=0
MOVL C01958 V=800.0 PL=0
MOVL C01959 V=800.0 PL=0
MOVL C01960 V=800.0 PL=0
MOVL C01961 V=800.0 PL=0
MOVL C01962 V=800.0 PL=0
MOVL C01963 V=800.0 PL=0
MOVL C01964 V=800.0 PL=0
MOVL C01965 V=800.0 PL=0
MOVL C01966 V=800.0 PL=0
MOVL C01967 V=800.0 PL=0
MOVL C01968 V=800.0 PL=0
MOVL C01969 V=800.0 PL=0
MOVL C01970 V=800.0 PL=0
MOVL C01971 V=800.0 PL=0
MOVL C01972 V=800.0 PL=0
MOVL C01973 V=800.0 PL=0
MOVL C01974 V=800.0 PL=0
MOVL C01975 V=800.0 PL=0
MOVL C01976 V=800.0 PL=0
MOVL C01977 V=800.0 PL=0
MOVL C01978 V=800.0 PL=0
MOVL C01979 V=800.0 PL=0
MOVL C01980 V=800.0 PL=0
MOVL C01981 V=800.0 PL=0
MOVL C01982 V=800.0 PL=0
MOVL C01983 V=800.0 PL=0
MOVL C01984 V=800.0 PL=0
MOVL C01985 V=800.0 PL=0
MOVL C01986 V=800.0 PL=0
MOVL C01987 V=800.0 PL=0
MOVL C01988 V=800.0 PL=0
MOVL C01989 V=800.0 PL=0
MOVL C01990 V=800.0 PL=0
MOVL C01991 V=800.0 PL=0
MOVL C01992 V=800.0 PL=0
MOVL C01993 V=800.0 PL=0
MOVL C01994 V=800.0 PL=0
MOVL C01995 V=800.0 PL=0
MOVL C01996 V=800.0 PL=0
MOVL C01997 V=800.0 PL=0
MOVL C01998 V=800.0 PL=0
MOVL C01999 V=800.0 PL=0
MOVL C02000 V=800.0 PL=0
MOVL C02001 V=800.0 PL=0
MOVL C02002 V=800.0 PL=0
MOVL C02003 V=800.0 PL=0
MOVL C02004 V=800.0 PL=0
MOVL C02005 V=800.0 PL=0
MOVL C02006 V=800.0 PL=0
MOVL C02007 V=800.0 PL=0
MOVL C02008 V=800.0 PL=0
MOVL C02009 V=800.0 PL=0
MOVL C02010 V=800.0 PL=0
MOVL C02011 V=800.0 PL=0
MOVL C02012 V=800.0 PL=0
MOVL C02013 V=800.0 PL=0
MOVL C02014 V=800.0 PL=0
MOVL C02015 V=800.0 PL=0
MOVL C02016 V=800.0 PL=0
MOVL C02017 V=800.0 PL=0
MOVL C02018 V=800.0 PL=0
MOVL C02019 V=800.0 PL=0
MOVL C02020 V=800.0 PL=0
MOVL C02021 V=800.0 PL=0
MOVL C02022 V=800.0 PL=0
MOVL C02023 V=800.0 PL=0
MOVL C02024 V=800.0 PL=0
MOVL C02025 V=800.0 PL=0
MOVL C02026 V=800.0 PL=0
MOVL C02027 V=800.0 PL=0
MOVL C02028 V=800.0 PL=0
MOVL C02029 V=800.0 PL=0
MOVL C02030 V=800.0 PL=0
MOVL C02031 V=800.0 PL=0
MOVL C02032 V=800.0 PL=0
MOVL C02033 V=800.0 PL=0
MOVL C02034 V=800.0 PL=0
MOVL C02035 V=800.0 PL=0
MOVL C02036 V=800.0 PL=0
MOVL C02037 V=800.0 PL=0
MOVL C02038 V=800.0 PL=0
MOVL C02039 V=800.0 PL=0
MOVL C02040 V=800.0 PL=0
MOVL C02041 V=800.0 PL=0
MOVL C02042 V=800.0 PL=0
MOVL C02043 V=800.0 PL=0
MOVL C02044 V=800.0 PL=0
MOVL C02045 V=800.0 PL=0
MOVL C02046 V=800.0 PL=0
MOVL C02047 V=800.0 PL=0
MOVL C02048 V=800.0 PL=0
MOVL C02049 V=800.0 PL=0
MOVL C02050 V=800.0 PL=0
MOVL C02051 V=800.0 PL=0
MOVL C02052 V=800.0 PL=0
MOVL C02053 V=800.0 PL=0
MOVL C02054 V=800.0 PL=0
MOVL C02055 V=800.0 PL=0
MOVL C02056 V=800.0 PL=0
MOVL C02057 V=800.0 PL=0
MOVL C02058 V=800.0 PL=0
MOVL C02059 V=800.0 PL=0
MOVL C02060 V=800.0 PL=0
MOVL C02061 V=800.0 PL=0
MOVL C02062 V=800.0 PL=0
MOVL C02063 V=800.0 PL=0
MOVL C02064 V=800.0 PL=0
MOVL C02065 V=800.0 PL=0
MOVL C02066 V=800.0 PL=0
MOVL C02067 V=800.0 PL=0
MOVL C02068 V=800.0 PL=0
MOVL C02069 V=800.0 PL=0
MOVL C02070 V=800.0 PL=0
MOVL C02071 V=800.0 PL=0
MOVL C02072 V=800.0 PL=0
MOVL C02073 V=800.0 PL=0
MOVL C02074 V=800.0 PL=0
MOVL C02075 V=800.0 PL=0
MOVL C02076 V=800.0 PL=0
MOVL C02077 V=800.0 PL=0
MOVL C02078 V=800.0 PL=0
MOVL C02079 V=800.0 PL=0
MOVL C02080 V=800.0 PL=0
MOVL C02081 V=800.0 PL=0
MOVL C02082 V=800.0 PL=0
MOVL C02083 V=800.0 PL=0
MOVL C02084 V=800.0 PL=0
MOVL C02085 V=800.0 PL=0
MOVL C02086 V=800.0 PL=0
MOVL C02087 V=800.0 PL=0
MOVL C02088 V=800.0 PL=0
MOVL C02089 V=800.0 PL=0
MOVL C02090 V=800.0 PL=0
MOVL C02091 V=800.0 PL=0
MOVL C02092 V=800.0 PL=0
MOVL C02093 V=800.0 PL=0
MOVL C02094 V=800.0 PL=0
MOVL C02095 V=800.0 PL=0
MOVL C02096 V=800.0 PL=0
MOVL C02097 V=800.0 PL=0
MOVL C02098 V=800.0 PL=0
MOVL C02099 V=800.0 PL=0
MOVL C02100 V=800.0 PL=0
MOVL C02101 V=800.0 PL=0
MOVL C02102 V=800.0 PL=0
MOVL C02103 V=800.0 PL=0
MOVL C02104 V=800.0 PL=0
MOVL C02105 V=800.0 PL=0
MOVL C02106 V=800.0 PL=0
MOVL C02107 V=800.0 PL=0
MOVL C02108 V=800.0 PL=0
MOVL C02109 V=800.0 PL=0
MOVL C02110 V=800.0 PL=0
MOVL C02111 V=800.0 PL=0
MOVL C02112 V=800.0 PL=0
MOVL C02113 V=800.0 PL=0
MOVL C02114 V=800.0 PL=0
MOVL C02115 V=800.0 PL=0
MOVL C02116 V=800.0 PL=0
MOVL C02117 V=800.0 PL=0
MOVL C02118 V=800.0 PL=0
MOVL C02119 V=800.0 PL=0
MOVL C02120 V=800.0 PL=0
MOVL C02121 V=800.0 PL=0
MOVL C02122 V=800.0 PL=0
MOVL C02123 V=800.0 PL=0
MOVL C02124 V=800.0 PL=0
MOVL C02125 V=800.0 PL=0
MOVL C02126 V=800.0 PL=0
MOVL C02127 V=800.0 PL=0
MOVL C02128 V=800.0 PL=0
MOVL C02129 V=800.0 PL=0
MOVL C02130 V=800.0 PL=0
MOVL C02131 V=800.0 PL=0
MOVL C02132 V=800.0 PL=0
MOVL C02133 V=800.0 PL=0
MOVL C02134 V=800.0 PL=0
MOVL C02135 V=800.0 PL=0
MOVL C02136 V=800.0 PL=0
MOVL C02137 V=800.0 PL=0
MOVL C02138 V=800.0 PL=0
MOVL C02139 V=800.0 PL=0
MOVL C02140 V=800.0 PL=0
MOVL C02141 V=800.0 PL=0
MOVL C02142 V=800.0 PL=0
MOVL C02143 V=800.0 PL=0
MOVL C02144 V=800.0 PL=0
MOVL C02145 V=800.0 PL=0
MOVL C02146 V=800.0 PL=0
MOVL C02147 V=800.0 PL=0
MOVL C02148 V=800.0 PL=0
MOVL C02149 V=800.0 PL=0
MOVL C02150 V=800.0 PL=0
MOVL C02151 V=800.0 PL=0
MOVL C02152 V=800.0 PL=0
MOVL C02153 V=800.0 PL=0
MOVL C02154 V=800.0 PL=0
MOVL C02155 V=800.0 PL=0
MOVL C02156 V=800.0 PL=0
MOVL C02157 V=800.0 PL=0
MOVL C02158 V=800.0 PL=0
MOVL C02159 V=800.0 PL=0
